// TIA Portal V17 export
// export: Created 2023-12-22T15:05:32.0644893Z, ExportSetting WithDefaults, DisplayName Totally Integrated Automation Portal, DisplayVersion V17, DisplayName TIA Portal Openness, DisplayVersion V17, DisplayName TIA Portal Version Control Interface, DisplayVersion V17, DisplayName STEP 7 Professional, DisplayVersion V17, DisplayName STEP 7 Safety, DisplayVersion V17, DisplayName WinCC Advanced, DisplayVersion V17
FUNCTION "ASCII_WCHAR_FC" : Void   // FC201, LAD
{ S7_Optimized_Access := 'TRUE' }
VERSION : 0.1
// stored: AutoNumber false, IsIECCheckEnabled false, SetENOAutomatically false, UDAEnableTagReadback false
   VAR_INPUT
      UNICODE : WChar;
   END_VAR
   VAR_OUTPUT
      ASCII_HEX : Byte;
   END_VAR
   VAR_IN_OUT
      DONE : Bool;
   END_VAR
BEGIN

REGION Network 1
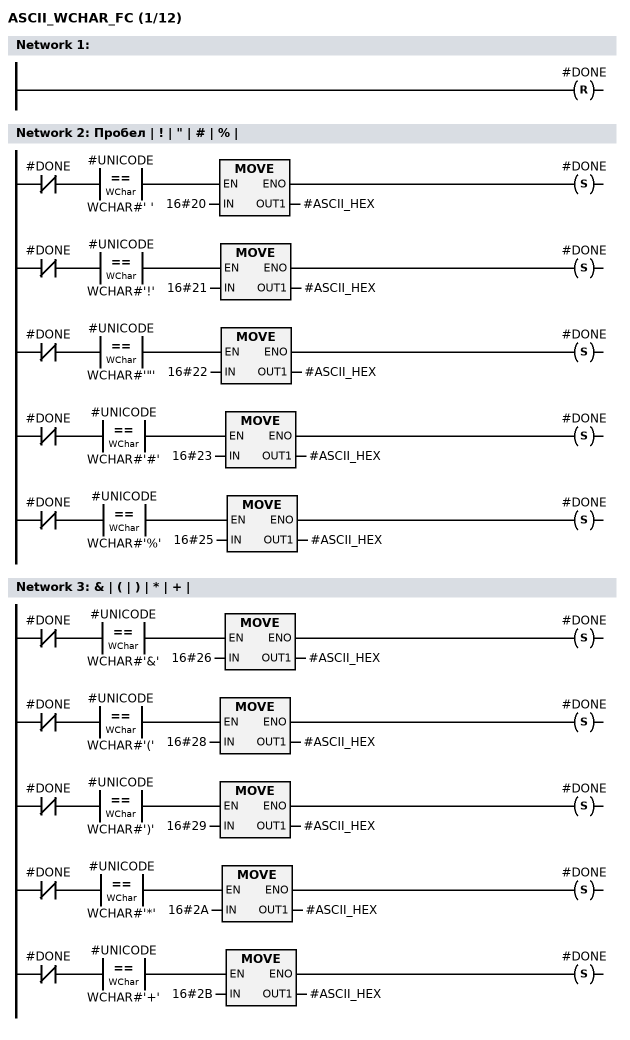
   RUNG wire#powerrail
      R_Coil( #DONE )
   END_RUNG
   // the same network as SCL:
   #DONE := FALSE;
END_REGION

REGION Network 2: Пробел | ! | " | # | % |
   RUNG wire#powerrail
      I_Contact( #DONE )
      { S7_Templates := "SrcType := WChar" } EQ_Contact(in1 := #UNICODE, in2 := WCHAR#' ')
      Move(in := 16#20, out1 => #ASCII_HEX)
      S_Coil( #DONE )
   END_RUNG
   RUNG wire#powerrail
      I_Contact( #DONE )
      { S7_Templates := "SrcType := WChar" } EQ_Contact(in1 := #UNICODE, in2 := WCHAR#'!')
      Move(in := 16#21, out1 => #ASCII_HEX)
      S_Coil( #DONE )
   END_RUNG
   RUNG wire#powerrail
      I_Contact( #DONE )
      { S7_Templates := "SrcType := WChar" } EQ_Contact(in1 := #UNICODE, in2 := WCHAR#'"')
      Move(in := 16#22, out1 => #ASCII_HEX)
      S_Coil( #DONE )
   END_RUNG
   RUNG wire#powerrail
      I_Contact( #DONE )
      { S7_Templates := "SrcType := WChar" } EQ_Contact(in1 := #UNICODE, in2 := WCHAR#'#')
      Move(in := 16#23, out1 => #ASCII_HEX)
      S_Coil( #DONE )
   END_RUNG
   RUNG wire#powerrail
      I_Contact( #DONE )
      { S7_Templates := "SrcType := WChar" } EQ_Contact(in1 := #UNICODE, in2 := WCHAR#'%')
      Move(in := 16#25, out1 => #ASCII_HEX)
      S_Coil( #DONE )
   END_RUNG
   // the same network as SCL:
   IF NOT #DONE AND (#UNICODE = WCHAR#' ') THEN
       #ASCII_HEX := 16#20;
       #DONE := TRUE;
   END_IF;
   IF NOT #DONE AND (#UNICODE = WCHAR#'!') THEN
       #ASCII_HEX := 16#21;
       #DONE := TRUE;
   END_IF;
   IF NOT #DONE AND (#UNICODE = WCHAR#'"') THEN
       #ASCII_HEX := 16#22;
       #DONE := TRUE;
   END_IF;
   IF NOT #DONE AND (#UNICODE = WCHAR#'#') THEN
       #ASCII_HEX := 16#23;
       #DONE := TRUE;
   END_IF;
   IF NOT #DONE AND (#UNICODE = WCHAR#'%') THEN
       #ASCII_HEX := 16#25;
       #DONE := TRUE;
   END_IF;
END_REGION

REGION Network 3: & | ( | ) | * | + |
   RUNG wire#powerrail
      I_Contact( #DONE )
      { S7_Templates := "SrcType := WChar" } EQ_Contact(in1 := #UNICODE, in2 := WCHAR#'&')
      Move(in := 16#26, out1 => #ASCII_HEX)
      S_Coil( #DONE )
   END_RUNG
   RUNG wire#powerrail
      I_Contact( #DONE )
      { S7_Templates := "SrcType := WChar" } EQ_Contact(in1 := #UNICODE, in2 := WCHAR#'(')
      Move(in := 16#28, out1 => #ASCII_HEX)
      S_Coil( #DONE )
   END_RUNG
   RUNG wire#powerrail
      I_Contact( #DONE )
      { S7_Templates := "SrcType := WChar" } EQ_Contact(in1 := #UNICODE, in2 := WCHAR#')')
      Move(in := 16#29, out1 => #ASCII_HEX)
      S_Coil( #DONE )
   END_RUNG
   RUNG wire#powerrail
      I_Contact( #DONE )
      { S7_Templates := "SrcType := WChar" } EQ_Contact(in1 := #UNICODE, in2 := WCHAR#'*')
      Move(in := 16#2A, out1 => #ASCII_HEX)
      S_Coil( #DONE )
   END_RUNG
   RUNG wire#powerrail
      I_Contact( #DONE )
      { S7_Templates := "SrcType := WChar" } EQ_Contact(in1 := #UNICODE, in2 := WCHAR#'+')
      Move(in := 16#2B, out1 => #ASCII_HEX)
      S_Coil( #DONE )
   END_RUNG
   // the same network as SCL:
   IF NOT #DONE AND (#UNICODE = WCHAR#'&') THEN
       #ASCII_HEX := 16#26;
       #DONE := TRUE;
   END_IF;
   IF NOT #DONE AND (#UNICODE = WCHAR#'(') THEN
       #ASCII_HEX := 16#28;
       #DONE := TRUE;
   END_IF;
   IF NOT #DONE AND (#UNICODE = WCHAR#')') THEN
       #ASCII_HEX := 16#29;
       #DONE := TRUE;
   END_IF;
   IF NOT #DONE AND (#UNICODE = WCHAR#'*') THEN
       #ASCII_HEX := 16#2A;
       #DONE := TRUE;
   END_IF;
   IF NOT #DONE AND (#UNICODE = WCHAR#'+') THEN
       #ASCII_HEX := 16#2B;
       #DONE := TRUE;
   END_IF;
END_REGION

REGION Network 4: , | - | . | / | : |
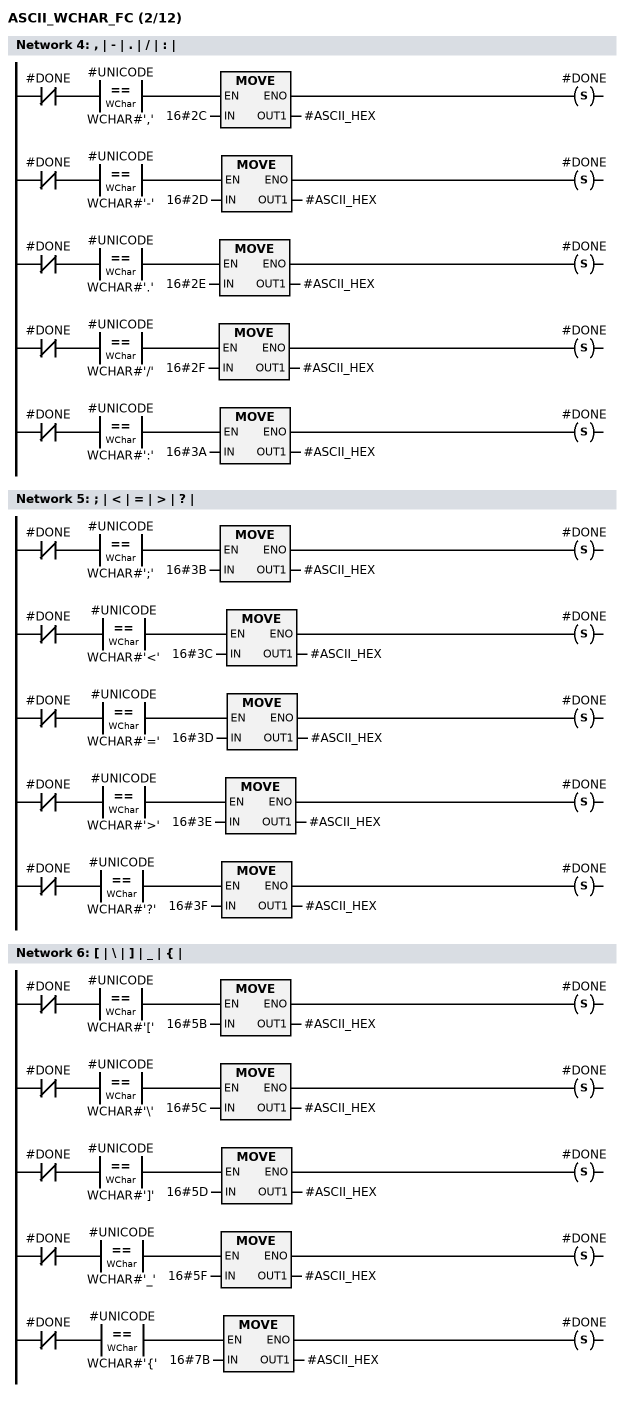
   RUNG wire#powerrail
      I_Contact( #DONE )
      { S7_Templates := "SrcType := WChar" } EQ_Contact(in1 := #UNICODE, in2 := WCHAR#',')
      Move(in := 16#2C, out1 => #ASCII_HEX)
      S_Coil( #DONE )
   END_RUNG
   RUNG wire#powerrail
      I_Contact( #DONE )
      { S7_Templates := "SrcType := WChar" } EQ_Contact(in1 := #UNICODE, in2 := WCHAR#'-')
      Move(in := 16#2D, out1 => #ASCII_HEX)
      S_Coil( #DONE )
   END_RUNG
   RUNG wire#powerrail
      I_Contact( #DONE )
      { S7_Templates := "SrcType := WChar" } EQ_Contact(in1 := #UNICODE, in2 := WCHAR#'.')
      Move(in := 16#2E, out1 => #ASCII_HEX)
      S_Coil( #DONE )
   END_RUNG
   RUNG wire#powerrail
      I_Contact( #DONE )
      { S7_Templates := "SrcType := WChar" } EQ_Contact(in1 := #UNICODE, in2 := WCHAR#'/')
      Move(in := 16#2F, out1 => #ASCII_HEX)
      S_Coil( #DONE )
   END_RUNG
   RUNG wire#powerrail
      I_Contact( #DONE )
      { S7_Templates := "SrcType := WChar" } EQ_Contact(in1 := #UNICODE, in2 := WCHAR#':')
      Move(in := 16#3A, out1 => #ASCII_HEX)
      S_Coil( #DONE )
   END_RUNG
   // the same network as SCL:
   IF NOT #DONE AND (#UNICODE = WCHAR#',') THEN
       #ASCII_HEX := 16#2C;
       #DONE := TRUE;
   END_IF;
   IF NOT #DONE AND (#UNICODE = WCHAR#'-') THEN
       #ASCII_HEX := 16#2D;
       #DONE := TRUE;
   END_IF;
   IF NOT #DONE AND (#UNICODE = WCHAR#'.') THEN
       #ASCII_HEX := 16#2E;
       #DONE := TRUE;
   END_IF;
   IF NOT #DONE AND (#UNICODE = WCHAR#'/') THEN
       #ASCII_HEX := 16#2F;
       #DONE := TRUE;
   END_IF;
   IF NOT #DONE AND (#UNICODE = WCHAR#':') THEN
       #ASCII_HEX := 16#3A;
       #DONE := TRUE;
   END_IF;
END_REGION

REGION Network 5: ; | < | = | > | ? |
   RUNG wire#powerrail
      I_Contact( #DONE )
      { S7_Templates := "SrcType := WChar" } EQ_Contact(in1 := #UNICODE, in2 := WCHAR#';')
      Move(in := 16#3B, out1 => #ASCII_HEX)
      S_Coil( #DONE )
   END_RUNG
   RUNG wire#powerrail
      I_Contact( #DONE )
      { S7_Templates := "SrcType := WChar" } EQ_Contact(in1 := #UNICODE, in2 := WCHAR#'<')
      Move(in := 16#3C, out1 => #ASCII_HEX)
      S_Coil( #DONE )
   END_RUNG
   RUNG wire#powerrail
      I_Contact( #DONE )
      { S7_Templates := "SrcType := WChar" } EQ_Contact(in1 := #UNICODE, in2 := WCHAR#'=')
      Move(in := 16#3D, out1 => #ASCII_HEX)
      S_Coil( #DONE )
   END_RUNG
   RUNG wire#powerrail
      I_Contact( #DONE )
      { S7_Templates := "SrcType := WChar" } EQ_Contact(in1 := #UNICODE, in2 := WCHAR#'>')
      Move(in := 16#3E, out1 => #ASCII_HEX)
      S_Coil( #DONE )
   END_RUNG
   RUNG wire#powerrail
      I_Contact( #DONE )
      { S7_Templates := "SrcType := WChar" } EQ_Contact(in1 := #UNICODE, in2 := WCHAR#'?')
      Move(in := 16#3F, out1 => #ASCII_HEX)
      S_Coil( #DONE )
   END_RUNG
   // the same network as SCL:
   IF NOT #DONE AND (#UNICODE = WCHAR#';') THEN
       #ASCII_HEX := 16#3B;
       #DONE := TRUE;
   END_IF;
   IF NOT #DONE AND (#UNICODE = WCHAR#'<') THEN
       #ASCII_HEX := 16#3C;
       #DONE := TRUE;
   END_IF;
   IF NOT #DONE AND (#UNICODE = WCHAR#'=') THEN
       #ASCII_HEX := 16#3D;
       #DONE := TRUE;
   END_IF;
   IF NOT #DONE AND (#UNICODE = WCHAR#'>') THEN
       #ASCII_HEX := 16#3E;
       #DONE := TRUE;
   END_IF;
   IF NOT #DONE AND (#UNICODE = WCHAR#'?') THEN
       #ASCII_HEX := 16#3F;
       #DONE := TRUE;
   END_IF;
END_REGION

REGION Network 6: [ | \ | ] | _ | { |
   RUNG wire#powerrail
      I_Contact( #DONE )
      { S7_Templates := "SrcType := WChar" } EQ_Contact(in1 := #UNICODE, in2 := WCHAR#'[')
      Move(in := 16#5B, out1 => #ASCII_HEX)
      S_Coil( #DONE )
   END_RUNG
   RUNG wire#powerrail
      I_Contact( #DONE )
      { S7_Templates := "SrcType := WChar" } EQ_Contact(in1 := #UNICODE, in2 := WCHAR#'\')
      Move(in := 16#5C, out1 => #ASCII_HEX)
      S_Coil( #DONE )
   END_RUNG
   RUNG wire#powerrail
      I_Contact( #DONE )
      { S7_Templates := "SrcType := WChar" } EQ_Contact(in1 := #UNICODE, in2 := WCHAR#']')
      Move(in := 16#5D, out1 => #ASCII_HEX)
      S_Coil( #DONE )
   END_RUNG
   RUNG wire#powerrail
      I_Contact( #DONE )
      { S7_Templates := "SrcType := WChar" } EQ_Contact(in1 := #UNICODE, in2 := WCHAR#'_')
      Move(in := 16#5F, out1 => #ASCII_HEX)
      S_Coil( #DONE )
   END_RUNG
   RUNG wire#powerrail
      I_Contact( #DONE )
      { S7_Templates := "SrcType := WChar" } EQ_Contact(in1 := #UNICODE, in2 := WCHAR#'{')
      Move(in := 16#7B, out1 => #ASCII_HEX)
      S_Coil( #DONE )
   END_RUNG
   // the same network as SCL:
   IF NOT #DONE AND (#UNICODE = WCHAR#'[') THEN
       #ASCII_HEX := 16#5B;
       #DONE := TRUE;
   END_IF;
   IF NOT #DONE AND (#UNICODE = WCHAR#'\') THEN
       #ASCII_HEX := 16#5C;
       #DONE := TRUE;
   END_IF;
   IF NOT #DONE AND (#UNICODE = WCHAR#']') THEN
       #ASCII_HEX := 16#5D;
       #DONE := TRUE;
   END_IF;
   IF NOT #DONE AND (#UNICODE = WCHAR#'_') THEN
       #ASCII_HEX := 16#5F;
       #DONE := TRUE;
   END_IF;
   IF NOT #DONE AND (#UNICODE = WCHAR#'{') THEN
       #ASCII_HEX := 16#7B;
       #DONE := TRUE;
   END_IF;
END_REGION

REGION Network 7: } | | |
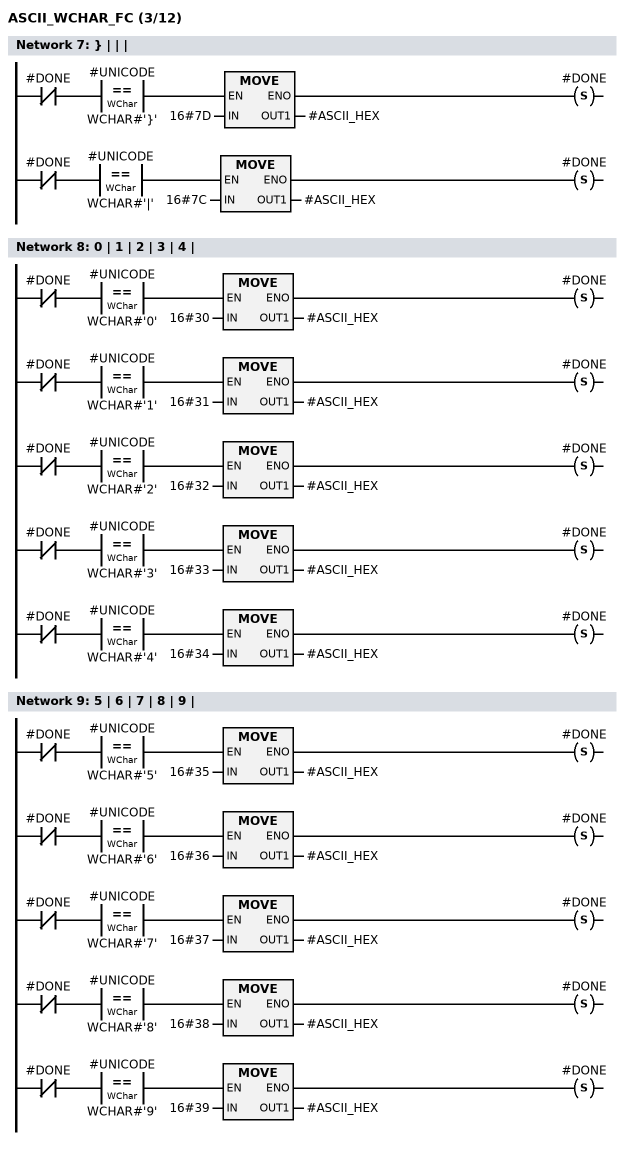
   RUNG wire#powerrail
      I_Contact( #DONE )
      { S7_Templates := "SrcType := WChar" } EQ_Contact(in1 := #UNICODE, in2 := WCHAR#'}')
      Move(in := 16#7D, out1 => #ASCII_HEX)
      S_Coil( #DONE )
   END_RUNG
   RUNG wire#powerrail
      I_Contact( #DONE )
      { S7_Templates := "SrcType := WChar" } EQ_Contact(in1 := #UNICODE, in2 := WCHAR#'|')
      Move(in := 16#7C, out1 => #ASCII_HEX)
      S_Coil( #DONE )
   END_RUNG
   // the same network as SCL:
   IF NOT #DONE AND (#UNICODE = WCHAR#'}') THEN
       #ASCII_HEX := 16#7D;
       #DONE := TRUE;
   END_IF;
   IF NOT #DONE AND (#UNICODE = WCHAR#'|') THEN
       #ASCII_HEX := 16#7C;
       #DONE := TRUE;
   END_IF;
END_REGION

REGION Network 8: 0 | 1 | 2 | 3 | 4 |
   RUNG wire#powerrail
      I_Contact( #DONE )
      { S7_Templates := "SrcType := WChar" } EQ_Contact(in1 := #UNICODE, in2 := WCHAR#'0')
      Move(in := 16#30, out1 => #ASCII_HEX)
      S_Coil( #DONE )
   END_RUNG
   RUNG wire#powerrail
      I_Contact( #DONE )
      { S7_Templates := "SrcType := WChar" } EQ_Contact(in1 := #UNICODE, in2 := WCHAR#'1')
      Move(in := 16#31, out1 => #ASCII_HEX)
      S_Coil( #DONE )
   END_RUNG
   RUNG wire#powerrail
      I_Contact( #DONE )
      { S7_Templates := "SrcType := WChar" } EQ_Contact(in1 := #UNICODE, in2 := WCHAR#'2')
      Move(in := 16#32, out1 => #ASCII_HEX)
      S_Coil( #DONE )
   END_RUNG
   RUNG wire#powerrail
      I_Contact( #DONE )
      { S7_Templates := "SrcType := WChar" } EQ_Contact(in1 := #UNICODE, in2 := WCHAR#'3')
      Move(in := 16#33, out1 => #ASCII_HEX)
      S_Coil( #DONE )
   END_RUNG
   RUNG wire#powerrail
      I_Contact( #DONE )
      { S7_Templates := "SrcType := WChar" } EQ_Contact(in1 := #UNICODE, in2 := WCHAR#'4')
      Move(in := 16#34, out1 => #ASCII_HEX)
      S_Coil( #DONE )
   END_RUNG
   // the same network as SCL:
   IF NOT #DONE AND (#UNICODE = WCHAR#'0') THEN
       #ASCII_HEX := 16#30;
       #DONE := TRUE;
   END_IF;
   IF NOT #DONE AND (#UNICODE = WCHAR#'1') THEN
       #ASCII_HEX := 16#31;
       #DONE := TRUE;
   END_IF;
   IF NOT #DONE AND (#UNICODE = WCHAR#'2') THEN
       #ASCII_HEX := 16#32;
       #DONE := TRUE;
   END_IF;
   IF NOT #DONE AND (#UNICODE = WCHAR#'3') THEN
       #ASCII_HEX := 16#33;
       #DONE := TRUE;
   END_IF;
   IF NOT #DONE AND (#UNICODE = WCHAR#'4') THEN
       #ASCII_HEX := 16#34;
       #DONE := TRUE;
   END_IF;
END_REGION

REGION Network 9: 5 | 6 | 7 | 8 | 9 |
   RUNG wire#powerrail
      I_Contact( #DONE )
      { S7_Templates := "SrcType := WChar" } EQ_Contact(in1 := #UNICODE, in2 := WCHAR#'5')
      Move(in := 16#35, out1 => #ASCII_HEX)
      S_Coil( #DONE )
   END_RUNG
   RUNG wire#powerrail
      I_Contact( #DONE )
      { S7_Templates := "SrcType := WChar" } EQ_Contact(in1 := #UNICODE, in2 := WCHAR#'6')
      Move(in := 16#36, out1 => #ASCII_HEX)
      S_Coil( #DONE )
   END_RUNG
   RUNG wire#powerrail
      I_Contact( #DONE )
      { S7_Templates := "SrcType := WChar" } EQ_Contact(in1 := #UNICODE, in2 := WCHAR#'7')
      Move(in := 16#37, out1 => #ASCII_HEX)
      S_Coil( #DONE )
   END_RUNG
   RUNG wire#powerrail
      I_Contact( #DONE )
      { S7_Templates := "SrcType := WChar" } EQ_Contact(in1 := #UNICODE, in2 := WCHAR#'8')
      Move(in := 16#38, out1 => #ASCII_HEX)
      S_Coil( #DONE )
   END_RUNG
   RUNG wire#powerrail
      I_Contact( #DONE )
      { S7_Templates := "SrcType := WChar" } EQ_Contact(in1 := #UNICODE, in2 := WCHAR#'9')
      Move(in := 16#39, out1 => #ASCII_HEX)
      S_Coil( #DONE )
   END_RUNG
   // the same network as SCL:
   IF NOT #DONE AND (#UNICODE = WCHAR#'5') THEN
       #ASCII_HEX := 16#35;
       #DONE := TRUE;
   END_IF;
   IF NOT #DONE AND (#UNICODE = WCHAR#'6') THEN
       #ASCII_HEX := 16#36;
       #DONE := TRUE;
   END_IF;
   IF NOT #DONE AND (#UNICODE = WCHAR#'7') THEN
       #ASCII_HEX := 16#37;
       #DONE := TRUE;
   END_IF;
   IF NOT #DONE AND (#UNICODE = WCHAR#'8') THEN
       #ASCII_HEX := 16#38;
       #DONE := TRUE;
   END_IF;
   IF NOT #DONE AND (#UNICODE = WCHAR#'9') THEN
       #ASCII_HEX := 16#39;
       #DONE := TRUE;
   END_IF;
END_REGION

REGION Network 10: А | Б | В | Г | Д |
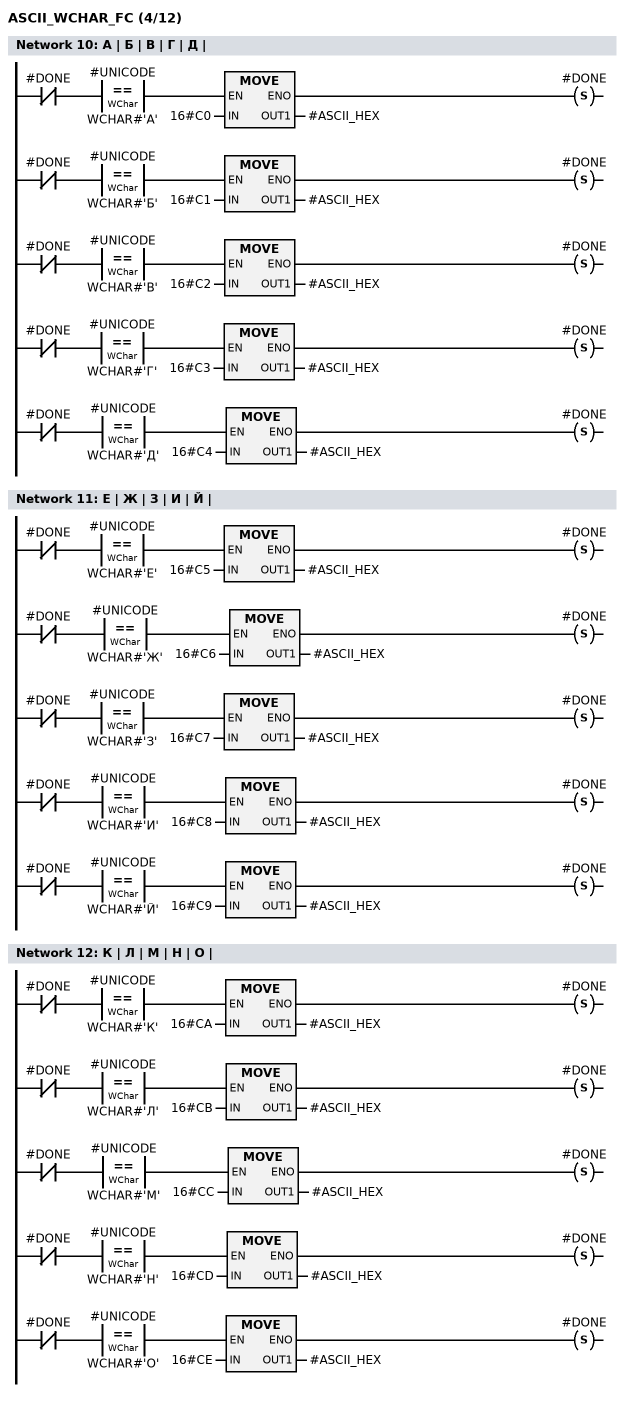
   RUNG wire#powerrail
      I_Contact( #DONE )
      { S7_Templates := "SrcType := WChar" } EQ_Contact(in1 := #UNICODE, in2 := WCHAR#'А')
      Move(in := 16#C0, out1 => #ASCII_HEX)
      S_Coil( #DONE )
   END_RUNG
   RUNG wire#powerrail
      I_Contact( #DONE )
      { S7_Templates := "SrcType := WChar" } EQ_Contact(in1 := #UNICODE, in2 := WCHAR#'Б')
      Move(in := 16#C1, out1 => #ASCII_HEX)
      S_Coil( #DONE )
   END_RUNG
   RUNG wire#powerrail
      I_Contact( #DONE )
      { S7_Templates := "SrcType := WChar" } EQ_Contact(in1 := #UNICODE, in2 := WCHAR#'В')
      Move(in := 16#C2, out1 => #ASCII_HEX)
      S_Coil( #DONE )
   END_RUNG
   RUNG wire#powerrail
      I_Contact( #DONE )
      { S7_Templates := "SrcType := WChar" } EQ_Contact(in1 := #UNICODE, in2 := WCHAR#'Г')
      Move(in := 16#C3, out1 => #ASCII_HEX)
      S_Coil( #DONE )
   END_RUNG
   RUNG wire#powerrail
      I_Contact( #DONE )
      { S7_Templates := "SrcType := WChar" } EQ_Contact(in1 := #UNICODE, in2 := WCHAR#'Д')
      Move(in := 16#C4, out1 => #ASCII_HEX)
      S_Coil( #DONE )
   END_RUNG
   // the same network as SCL:
   IF NOT #DONE AND (#UNICODE = WCHAR#'А') THEN
       #ASCII_HEX := 16#C0;
       #DONE := TRUE;
   END_IF;
   IF NOT #DONE AND (#UNICODE = WCHAR#'Б') THEN
       #ASCII_HEX := 16#C1;
       #DONE := TRUE;
   END_IF;
   IF NOT #DONE AND (#UNICODE = WCHAR#'В') THEN
       #ASCII_HEX := 16#C2;
       #DONE := TRUE;
   END_IF;
   IF NOT #DONE AND (#UNICODE = WCHAR#'Г') THEN
       #ASCII_HEX := 16#C3;
       #DONE := TRUE;
   END_IF;
   IF NOT #DONE AND (#UNICODE = WCHAR#'Д') THEN
       #ASCII_HEX := 16#C4;
       #DONE := TRUE;
   END_IF;
END_REGION

REGION Network 11: Е | Ж | З | И | Й |
   RUNG wire#powerrail
      I_Contact( #DONE )
      { S7_Templates := "SrcType := WChar" } EQ_Contact(in1 := #UNICODE, in2 := WCHAR#'Е')
      Move(in := 16#C5, out1 => #ASCII_HEX)
      S_Coil( #DONE )
   END_RUNG
   RUNG wire#powerrail
      I_Contact( #DONE )
      { S7_Templates := "SrcType := WChar" } EQ_Contact(in1 := #UNICODE, in2 := WCHAR#'Ж')
      Move(in := 16#C6, out1 => #ASCII_HEX)
      S_Coil( #DONE )
   END_RUNG
   RUNG wire#powerrail
      I_Contact( #DONE )
      { S7_Templates := "SrcType := WChar" } EQ_Contact(in1 := #UNICODE, in2 := WCHAR#'З')
      Move(in := 16#C7, out1 => #ASCII_HEX)
      S_Coil( #DONE )
   END_RUNG
   RUNG wire#powerrail
      I_Contact( #DONE )
      { S7_Templates := "SrcType := WChar" } EQ_Contact(in1 := #UNICODE, in2 := WCHAR#'И')
      Move(in := 16#C8, out1 => #ASCII_HEX)
      S_Coil( #DONE )
   END_RUNG
   RUNG wire#powerrail
      I_Contact( #DONE )
      { S7_Templates := "SrcType := WChar" } EQ_Contact(in1 := #UNICODE, in2 := WCHAR#'Й')
      Move(in := 16#C9, out1 => #ASCII_HEX)
      S_Coil( #DONE )
   END_RUNG
   // the same network as SCL:
   IF NOT #DONE AND (#UNICODE = WCHAR#'Е') THEN
       #ASCII_HEX := 16#C5;
       #DONE := TRUE;
   END_IF;
   IF NOT #DONE AND (#UNICODE = WCHAR#'Ж') THEN
       #ASCII_HEX := 16#C6;
       #DONE := TRUE;
   END_IF;
   IF NOT #DONE AND (#UNICODE = WCHAR#'З') THEN
       #ASCII_HEX := 16#C7;
       #DONE := TRUE;
   END_IF;
   IF NOT #DONE AND (#UNICODE = WCHAR#'И') THEN
       #ASCII_HEX := 16#C8;
       #DONE := TRUE;
   END_IF;
   IF NOT #DONE AND (#UNICODE = WCHAR#'Й') THEN
       #ASCII_HEX := 16#C9;
       #DONE := TRUE;
   END_IF;
END_REGION

REGION Network 12: К | Л | М | Н | О |
   RUNG wire#powerrail
      I_Contact( #DONE )
      { S7_Templates := "SrcType := WChar" } EQ_Contact(in1 := #UNICODE, in2 := WCHAR#'К')
      Move(in := 16#CA, out1 => #ASCII_HEX)
      S_Coil( #DONE )
   END_RUNG
   RUNG wire#powerrail
      I_Contact( #DONE )
      { S7_Templates := "SrcType := WChar" } EQ_Contact(in1 := #UNICODE, in2 := WCHAR#'Л')
      Move(in := 16#CB, out1 => #ASCII_HEX)
      S_Coil( #DONE )
   END_RUNG
   RUNG wire#powerrail
      I_Contact( #DONE )
      { S7_Templates := "SrcType := WChar" } EQ_Contact(in1 := #UNICODE, in2 := WCHAR#'М')
      Move(in := 16#CC, out1 => #ASCII_HEX)
      S_Coil( #DONE )
   END_RUNG
   RUNG wire#powerrail
      I_Contact( #DONE )
      { S7_Templates := "SrcType := WChar" } EQ_Contact(in1 := #UNICODE, in2 := WCHAR#'Н')
      Move(in := 16#CD, out1 => #ASCII_HEX)
      S_Coil( #DONE )
   END_RUNG
   RUNG wire#powerrail
      I_Contact( #DONE )
      { S7_Templates := "SrcType := WChar" } EQ_Contact(in1 := #UNICODE, in2 := WCHAR#'О')
      Move(in := 16#CE, out1 => #ASCII_HEX)
      S_Coil( #DONE )
   END_RUNG
   // the same network as SCL:
   IF NOT #DONE AND (#UNICODE = WCHAR#'К') THEN
       #ASCII_HEX := 16#CA;
       #DONE := TRUE;
   END_IF;
   IF NOT #DONE AND (#UNICODE = WCHAR#'Л') THEN
       #ASCII_HEX := 16#CB;
       #DONE := TRUE;
   END_IF;
   IF NOT #DONE AND (#UNICODE = WCHAR#'М') THEN
       #ASCII_HEX := 16#CC;
       #DONE := TRUE;
   END_IF;
   IF NOT #DONE AND (#UNICODE = WCHAR#'Н') THEN
       #ASCII_HEX := 16#CD;
       #DONE := TRUE;
   END_IF;
   IF NOT #DONE AND (#UNICODE = WCHAR#'О') THEN
       #ASCII_HEX := 16#CE;
       #DONE := TRUE;
   END_IF;
END_REGION

REGION Network 13: П | Р | С | Т | У |
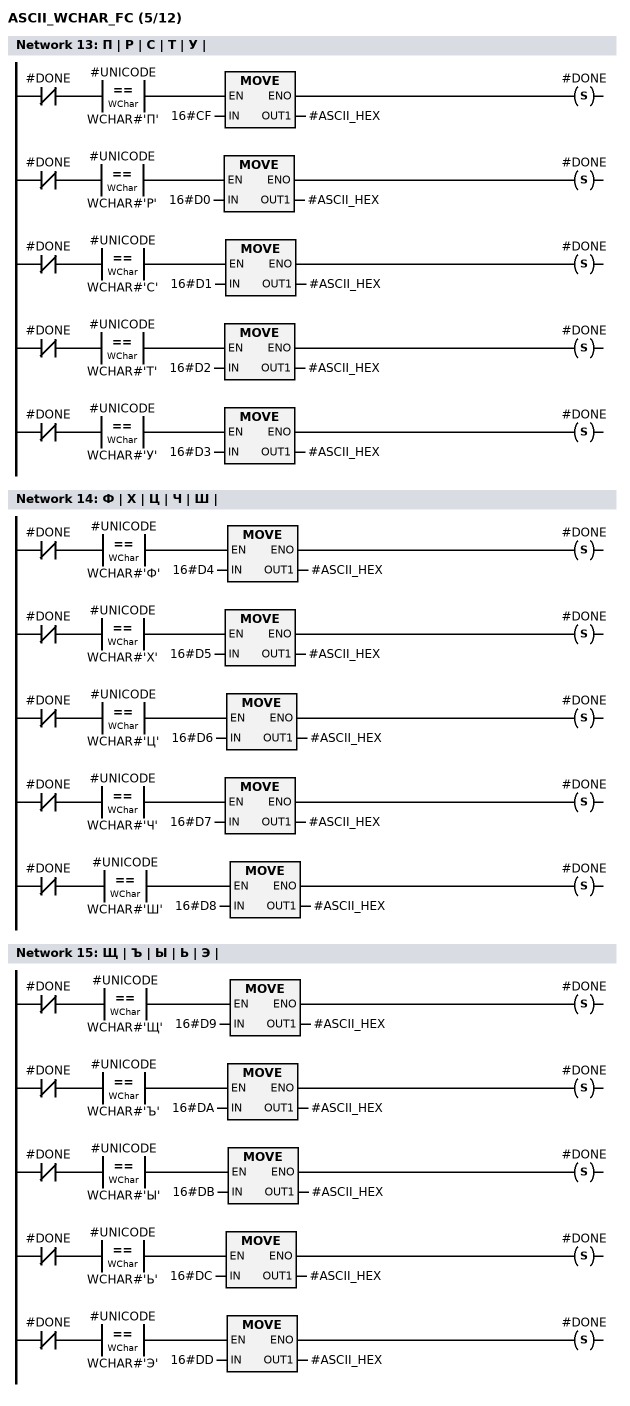
   RUNG wire#powerrail
      I_Contact( #DONE )
      { S7_Templates := "SrcType := WChar" } EQ_Contact(in1 := #UNICODE, in2 := WCHAR#'П')
      Move(in := 16#CF, out1 => #ASCII_HEX)
      S_Coil( #DONE )
   END_RUNG
   RUNG wire#powerrail
      I_Contact( #DONE )
      { S7_Templates := "SrcType := WChar" } EQ_Contact(in1 := #UNICODE, in2 := WCHAR#'Р')
      Move(in := 16#D0, out1 => #ASCII_HEX)
      S_Coil( #DONE )
   END_RUNG
   RUNG wire#powerrail
      I_Contact( #DONE )
      { S7_Templates := "SrcType := WChar" } EQ_Contact(in1 := #UNICODE, in2 := WCHAR#'С')
      Move(in := 16#D1, out1 => #ASCII_HEX)
      S_Coil( #DONE )
   END_RUNG
   RUNG wire#powerrail
      I_Contact( #DONE )
      { S7_Templates := "SrcType := WChar" } EQ_Contact(in1 := #UNICODE, in2 := WCHAR#'Т')
      Move(in := 16#D2, out1 => #ASCII_HEX)
      S_Coil( #DONE )
   END_RUNG
   RUNG wire#powerrail
      I_Contact( #DONE )
      { S7_Templates := "SrcType := WChar" } EQ_Contact(in1 := #UNICODE, in2 := WCHAR#'У')
      Move(in := 16#D3, out1 => #ASCII_HEX)
      S_Coil( #DONE )
   END_RUNG
   // the same network as SCL:
   IF NOT #DONE AND (#UNICODE = WCHAR#'П') THEN
       #ASCII_HEX := 16#CF;
       #DONE := TRUE;
   END_IF;
   IF NOT #DONE AND (#UNICODE = WCHAR#'Р') THEN
       #ASCII_HEX := 16#D0;
       #DONE := TRUE;
   END_IF;
   IF NOT #DONE AND (#UNICODE = WCHAR#'С') THEN
       #ASCII_HEX := 16#D1;
       #DONE := TRUE;
   END_IF;
   IF NOT #DONE AND (#UNICODE = WCHAR#'Т') THEN
       #ASCII_HEX := 16#D2;
       #DONE := TRUE;
   END_IF;
   IF NOT #DONE AND (#UNICODE = WCHAR#'У') THEN
       #ASCII_HEX := 16#D3;
       #DONE := TRUE;
   END_IF;
END_REGION

REGION Network 14: Ф | Х | Ц | Ч | Ш |
   RUNG wire#powerrail
      I_Contact( #DONE )
      { S7_Templates := "SrcType := WChar" } EQ_Contact(in1 := #UNICODE, in2 := WCHAR#'Ф')
      Move(in := 16#D4, out1 => #ASCII_HEX)
      S_Coil( #DONE )
   END_RUNG
   RUNG wire#powerrail
      I_Contact( #DONE )
      { S7_Templates := "SrcType := WChar" } EQ_Contact(in1 := #UNICODE, in2 := WCHAR#'Х')
      Move(in := 16#D5, out1 => #ASCII_HEX)
      S_Coil( #DONE )
   END_RUNG
   RUNG wire#powerrail
      I_Contact( #DONE )
      { S7_Templates := "SrcType := WChar" } EQ_Contact(in1 := #UNICODE, in2 := WCHAR#'Ц')
      Move(in := 16#D6, out1 => #ASCII_HEX)
      S_Coil( #DONE )
   END_RUNG
   RUNG wire#powerrail
      I_Contact( #DONE )
      { S7_Templates := "SrcType := WChar" } EQ_Contact(in1 := #UNICODE, in2 := WCHAR#'Ч')
      Move(in := 16#D7, out1 => #ASCII_HEX)
      S_Coil( #DONE )
   END_RUNG
   RUNG wire#powerrail
      I_Contact( #DONE )
      { S7_Templates := "SrcType := WChar" } EQ_Contact(in1 := #UNICODE, in2 := WCHAR#'Ш')
      Move(in := 16#D8, out1 => #ASCII_HEX)
      S_Coil( #DONE )
   END_RUNG
   // the same network as SCL:
   IF NOT #DONE AND (#UNICODE = WCHAR#'Ф') THEN
       #ASCII_HEX := 16#D4;
       #DONE := TRUE;
   END_IF;
   IF NOT #DONE AND (#UNICODE = WCHAR#'Х') THEN
       #ASCII_HEX := 16#D5;
       #DONE := TRUE;
   END_IF;
   IF NOT #DONE AND (#UNICODE = WCHAR#'Ц') THEN
       #ASCII_HEX := 16#D6;
       #DONE := TRUE;
   END_IF;
   IF NOT #DONE AND (#UNICODE = WCHAR#'Ч') THEN
       #ASCII_HEX := 16#D7;
       #DONE := TRUE;
   END_IF;
   IF NOT #DONE AND (#UNICODE = WCHAR#'Ш') THEN
       #ASCII_HEX := 16#D8;
       #DONE := TRUE;
   END_IF;
END_REGION

REGION Network 15: Щ | Ъ | Ы | Ь | Э |
   RUNG wire#powerrail
      I_Contact( #DONE )
      { S7_Templates := "SrcType := WChar" } EQ_Contact(in1 := #UNICODE, in2 := WCHAR#'Щ')
      Move(in := 16#D9, out1 => #ASCII_HEX)
      S_Coil( #DONE )
   END_RUNG
   RUNG wire#powerrail
      I_Contact( #DONE )
      { S7_Templates := "SrcType := WChar" } EQ_Contact(in1 := #UNICODE, in2 := WCHAR#'Ъ')
      Move(in := 16#DA, out1 => #ASCII_HEX)
      S_Coil( #DONE )
   END_RUNG
   RUNG wire#powerrail
      I_Contact( #DONE )
      { S7_Templates := "SrcType := WChar" } EQ_Contact(in1 := #UNICODE, in2 := WCHAR#'Ы')
      Move(in := 16#DB, out1 => #ASCII_HEX)
      S_Coil( #DONE )
   END_RUNG
   RUNG wire#powerrail
      I_Contact( #DONE )
      { S7_Templates := "SrcType := WChar" } EQ_Contact(in1 := #UNICODE, in2 := WCHAR#'Ь')
      Move(in := 16#DC, out1 => #ASCII_HEX)
      S_Coil( #DONE )
   END_RUNG
   RUNG wire#powerrail
      I_Contact( #DONE )
      { S7_Templates := "SrcType := WChar" } EQ_Contact(in1 := #UNICODE, in2 := WCHAR#'Э')
      Move(in := 16#DD, out1 => #ASCII_HEX)
      S_Coil( #DONE )
   END_RUNG
   // the same network as SCL:
   IF NOT #DONE AND (#UNICODE = WCHAR#'Щ') THEN
       #ASCII_HEX := 16#D9;
       #DONE := TRUE;
   END_IF;
   IF NOT #DONE AND (#UNICODE = WCHAR#'Ъ') THEN
       #ASCII_HEX := 16#DA;
       #DONE := TRUE;
   END_IF;
   IF NOT #DONE AND (#UNICODE = WCHAR#'Ы') THEN
       #ASCII_HEX := 16#DB;
       #DONE := TRUE;
   END_IF;
   IF NOT #DONE AND (#UNICODE = WCHAR#'Ь') THEN
       #ASCII_HEX := 16#DC;
       #DONE := TRUE;
   END_IF;
   IF NOT #DONE AND (#UNICODE = WCHAR#'Э') THEN
       #ASCII_HEX := 16#DD;
       #DONE := TRUE;
   END_IF;
END_REGION

REGION Network 16: Ю | Я |
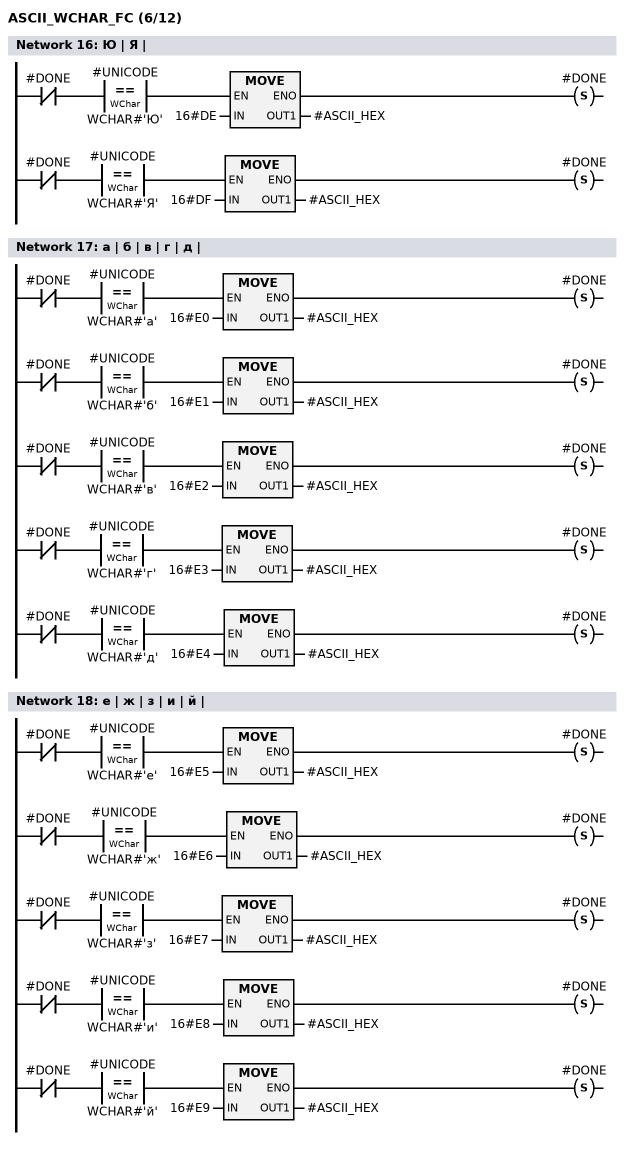
   RUNG wire#powerrail
      I_Contact( #DONE )
      { S7_Templates := "SrcType := WChar" } EQ_Contact(in1 := #UNICODE, in2 := WCHAR#'Ю')
      Move(in := 16#DE, out1 => #ASCII_HEX)
      S_Coil( #DONE )
   END_RUNG
   RUNG wire#powerrail
      I_Contact( #DONE )
      { S7_Templates := "SrcType := WChar" } EQ_Contact(in1 := #UNICODE, in2 := WCHAR#'Я')
      Move(in := 16#DF, out1 => #ASCII_HEX)
      S_Coil( #DONE )
   END_RUNG
   // the same network as SCL:
   IF NOT #DONE AND (#UNICODE = WCHAR#'Ю') THEN
       #ASCII_HEX := 16#DE;
       #DONE := TRUE;
   END_IF;
   IF NOT #DONE AND (#UNICODE = WCHAR#'Я') THEN
       #ASCII_HEX := 16#DF;
       #DONE := TRUE;
   END_IF;
END_REGION

REGION Network 17: а | б | в | г | д |
   RUNG wire#powerrail
      I_Contact( #DONE )
      { S7_Templates := "SrcType := WChar" } EQ_Contact(in1 := #UNICODE, in2 := WCHAR#'а')
      Move(in := 16#E0, out1 => #ASCII_HEX)
      S_Coil( #DONE )
   END_RUNG
   RUNG wire#powerrail
      I_Contact( #DONE )
      { S7_Templates := "SrcType := WChar" } EQ_Contact(in1 := #UNICODE, in2 := WCHAR#'б')
      Move(in := 16#E1, out1 => #ASCII_HEX)
      S_Coil( #DONE )
   END_RUNG
   RUNG wire#powerrail
      I_Contact( #DONE )
      { S7_Templates := "SrcType := WChar" } EQ_Contact(in1 := #UNICODE, in2 := WCHAR#'в')
      Move(in := 16#E2, out1 => #ASCII_HEX)
      S_Coil( #DONE )
   END_RUNG
   RUNG wire#powerrail
      I_Contact( #DONE )
      { S7_Templates := "SrcType := WChar" } EQ_Contact(in1 := #UNICODE, in2 := WCHAR#'г')
      Move(in := 16#E3, out1 => #ASCII_HEX)
      S_Coil( #DONE )
   END_RUNG
   RUNG wire#powerrail
      I_Contact( #DONE )
      { S7_Templates := "SrcType := WChar" } EQ_Contact(in1 := #UNICODE, in2 := WCHAR#'д')
      Move(in := 16#E4, out1 => #ASCII_HEX)
      S_Coil( #DONE )
   END_RUNG
   // the same network as SCL:
   IF NOT #DONE AND (#UNICODE = WCHAR#'а') THEN
       #ASCII_HEX := 16#E0;
       #DONE := TRUE;
   END_IF;
   IF NOT #DONE AND (#UNICODE = WCHAR#'б') THEN
       #ASCII_HEX := 16#E1;
       #DONE := TRUE;
   END_IF;
   IF NOT #DONE AND (#UNICODE = WCHAR#'в') THEN
       #ASCII_HEX := 16#E2;
       #DONE := TRUE;
   END_IF;
   IF NOT #DONE AND (#UNICODE = WCHAR#'г') THEN
       #ASCII_HEX := 16#E3;
       #DONE := TRUE;
   END_IF;
   IF NOT #DONE AND (#UNICODE = WCHAR#'д') THEN
       #ASCII_HEX := 16#E4;
       #DONE := TRUE;
   END_IF;
END_REGION

REGION Network 18: е | ж | з | и | й |
   RUNG wire#powerrail
      I_Contact( #DONE )
      { S7_Templates := "SrcType := WChar" } EQ_Contact(in1 := #UNICODE, in2 := WCHAR#'е')
      Move(in := 16#E5, out1 => #ASCII_HEX)
      S_Coil( #DONE )
   END_RUNG
   RUNG wire#powerrail
      I_Contact( #DONE )
      { S7_Templates := "SrcType := WChar" } EQ_Contact(in1 := #UNICODE, in2 := WCHAR#'ж')
      Move(in := 16#E6, out1 => #ASCII_HEX)
      S_Coil( #DONE )
   END_RUNG
   RUNG wire#powerrail
      I_Contact( #DONE )
      { S7_Templates := "SrcType := WChar" } EQ_Contact(in1 := #UNICODE, in2 := WCHAR#'з')
      Move(in := 16#E7, out1 => #ASCII_HEX)
      S_Coil( #DONE )
   END_RUNG
   RUNG wire#powerrail
      I_Contact( #DONE )
      { S7_Templates := "SrcType := WChar" } EQ_Contact(in1 := #UNICODE, in2 := WCHAR#'и')
      Move(in := 16#E8, out1 => #ASCII_HEX)
      S_Coil( #DONE )
   END_RUNG
   RUNG wire#powerrail
      I_Contact( #DONE )
      { S7_Templates := "SrcType := WChar" } EQ_Contact(in1 := #UNICODE, in2 := WCHAR#'й')
      Move(in := 16#E9, out1 => #ASCII_HEX)
      S_Coil( #DONE )
   END_RUNG
   // the same network as SCL:
   IF NOT #DONE AND (#UNICODE = WCHAR#'е') THEN
       #ASCII_HEX := 16#E5;
       #DONE := TRUE;
   END_IF;
   IF NOT #DONE AND (#UNICODE = WCHAR#'ж') THEN
       #ASCII_HEX := 16#E6;
       #DONE := TRUE;
   END_IF;
   IF NOT #DONE AND (#UNICODE = WCHAR#'з') THEN
       #ASCII_HEX := 16#E7;
       #DONE := TRUE;
   END_IF;
   IF NOT #DONE AND (#UNICODE = WCHAR#'и') THEN
       #ASCII_HEX := 16#E8;
       #DONE := TRUE;
   END_IF;
   IF NOT #DONE AND (#UNICODE = WCHAR#'й') THEN
       #ASCII_HEX := 16#E9;
       #DONE := TRUE;
   END_IF;
END_REGION

REGION Network 19: к | л | м | н | о |
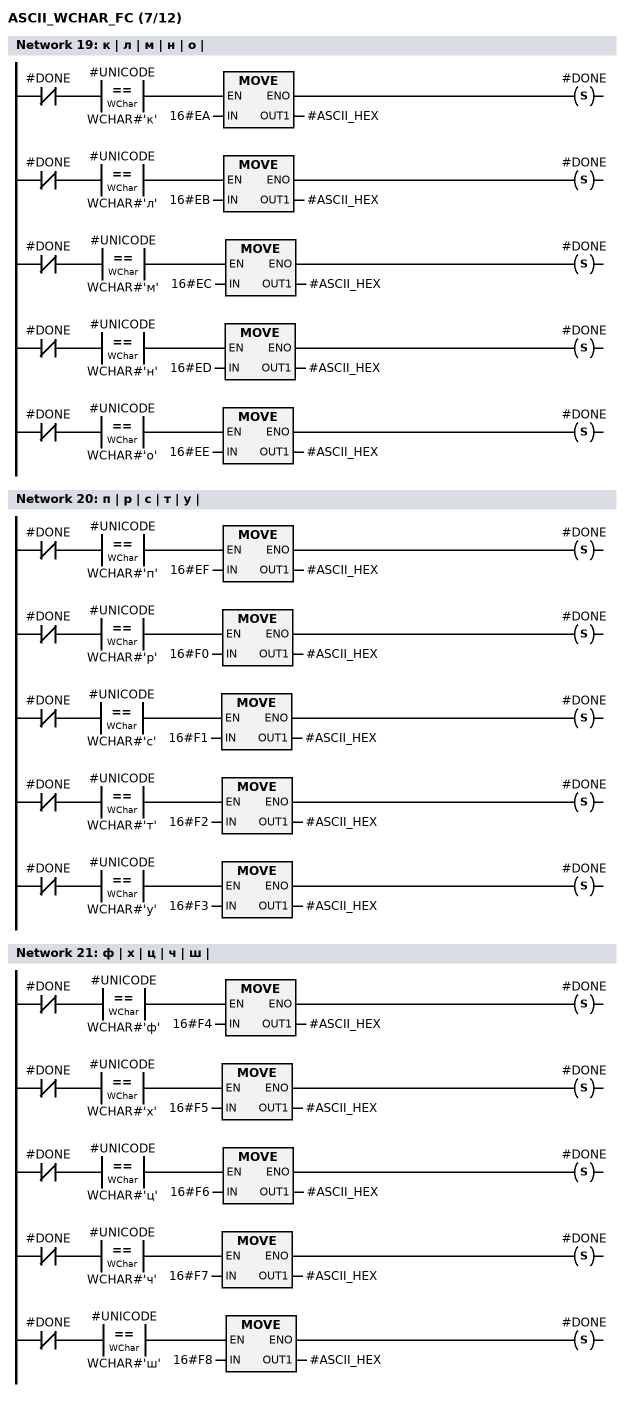
   RUNG wire#powerrail
      I_Contact( #DONE )
      { S7_Templates := "SrcType := WChar" } EQ_Contact(in1 := #UNICODE, in2 := WCHAR#'к')
      Move(in := 16#EA, out1 => #ASCII_HEX)
      S_Coil( #DONE )
   END_RUNG
   RUNG wire#powerrail
      I_Contact( #DONE )
      { S7_Templates := "SrcType := WChar" } EQ_Contact(in1 := #UNICODE, in2 := WCHAR#'л')
      Move(in := 16#EB, out1 => #ASCII_HEX)
      S_Coil( #DONE )
   END_RUNG
   RUNG wire#powerrail
      I_Contact( #DONE )
      { S7_Templates := "SrcType := WChar" } EQ_Contact(in1 := #UNICODE, in2 := WCHAR#'м')
      Move(in := 16#EC, out1 => #ASCII_HEX)
      S_Coil( #DONE )
   END_RUNG
   RUNG wire#powerrail
      I_Contact( #DONE )
      { S7_Templates := "SrcType := WChar" } EQ_Contact(in1 := #UNICODE, in2 := WCHAR#'н')
      Move(in := 16#ED, out1 => #ASCII_HEX)
      S_Coil( #DONE )
   END_RUNG
   RUNG wire#powerrail
      I_Contact( #DONE )
      { S7_Templates := "SrcType := WChar" } EQ_Contact(in1 := #UNICODE, in2 := WCHAR#'о')
      Move(in := 16#EE, out1 => #ASCII_HEX)
      S_Coil( #DONE )
   END_RUNG
   // the same network as SCL:
   IF NOT #DONE AND (#UNICODE = WCHAR#'к') THEN
       #ASCII_HEX := 16#EA;
       #DONE := TRUE;
   END_IF;
   IF NOT #DONE AND (#UNICODE = WCHAR#'л') THEN
       #ASCII_HEX := 16#EB;
       #DONE := TRUE;
   END_IF;
   IF NOT #DONE AND (#UNICODE = WCHAR#'м') THEN
       #ASCII_HEX := 16#EC;
       #DONE := TRUE;
   END_IF;
   IF NOT #DONE AND (#UNICODE = WCHAR#'н') THEN
       #ASCII_HEX := 16#ED;
       #DONE := TRUE;
   END_IF;
   IF NOT #DONE AND (#UNICODE = WCHAR#'о') THEN
       #ASCII_HEX := 16#EE;
       #DONE := TRUE;
   END_IF;
END_REGION

REGION Network 20: п | р | с | т | у |
   RUNG wire#powerrail
      I_Contact( #DONE )
      { S7_Templates := "SrcType := WChar" } EQ_Contact(in1 := #UNICODE, in2 := WCHAR#'п')
      Move(in := 16#EF, out1 => #ASCII_HEX)
      S_Coil( #DONE )
   END_RUNG
   RUNG wire#powerrail
      I_Contact( #DONE )
      { S7_Templates := "SrcType := WChar" } EQ_Contact(in1 := #UNICODE, in2 := WCHAR#'р')
      Move(in := 16#F0, out1 => #ASCII_HEX)
      S_Coil( #DONE )
   END_RUNG
   RUNG wire#powerrail
      I_Contact( #DONE )
      { S7_Templates := "SrcType := WChar" } EQ_Contact(in1 := #UNICODE, in2 := WCHAR#'с')
      Move(in := 16#F1, out1 => #ASCII_HEX)
      S_Coil( #DONE )
   END_RUNG
   RUNG wire#powerrail
      I_Contact( #DONE )
      { S7_Templates := "SrcType := WChar" } EQ_Contact(in1 := #UNICODE, in2 := WCHAR#'т')
      Move(in := 16#F2, out1 => #ASCII_HEX)
      S_Coil( #DONE )
   END_RUNG
   RUNG wire#powerrail
      I_Contact( #DONE )
      { S7_Templates := "SrcType := WChar" } EQ_Contact(in1 := #UNICODE, in2 := WCHAR#'у')
      Move(in := 16#F3, out1 => #ASCII_HEX)
      S_Coil( #DONE )
   END_RUNG
   // the same network as SCL:
   IF NOT #DONE AND (#UNICODE = WCHAR#'п') THEN
       #ASCII_HEX := 16#EF;
       #DONE := TRUE;
   END_IF;
   IF NOT #DONE AND (#UNICODE = WCHAR#'р') THEN
       #ASCII_HEX := 16#F0;
       #DONE := TRUE;
   END_IF;
   IF NOT #DONE AND (#UNICODE = WCHAR#'с') THEN
       #ASCII_HEX := 16#F1;
       #DONE := TRUE;
   END_IF;
   IF NOT #DONE AND (#UNICODE = WCHAR#'т') THEN
       #ASCII_HEX := 16#F2;
       #DONE := TRUE;
   END_IF;
   IF NOT #DONE AND (#UNICODE = WCHAR#'у') THEN
       #ASCII_HEX := 16#F3;
       #DONE := TRUE;
   END_IF;
END_REGION

REGION Network 21: ф | х | ц | ч | ш |
   RUNG wire#powerrail
      I_Contact( #DONE )
      { S7_Templates := "SrcType := WChar" } EQ_Contact(in1 := #UNICODE, in2 := WCHAR#'ф')
      Move(in := 16#F4, out1 => #ASCII_HEX)
      S_Coil( #DONE )
   END_RUNG
   RUNG wire#powerrail
      I_Contact( #DONE )
      { S7_Templates := "SrcType := WChar" } EQ_Contact(in1 := #UNICODE, in2 := WCHAR#'х')
      Move(in := 16#F5, out1 => #ASCII_HEX)
      S_Coil( #DONE )
   END_RUNG
   RUNG wire#powerrail
      I_Contact( #DONE )
      { S7_Templates := "SrcType := WChar" } EQ_Contact(in1 := #UNICODE, in2 := WCHAR#'ц')
      Move(in := 16#F6, out1 => #ASCII_HEX)
      S_Coil( #DONE )
   END_RUNG
   RUNG wire#powerrail
      I_Contact( #DONE )
      { S7_Templates := "SrcType := WChar" } EQ_Contact(in1 := #UNICODE, in2 := WCHAR#'ч')
      Move(in := 16#F7, out1 => #ASCII_HEX)
      S_Coil( #DONE )
   END_RUNG
   RUNG wire#powerrail
      I_Contact( #DONE )
      { S7_Templates := "SrcType := WChar" } EQ_Contact(in1 := #UNICODE, in2 := WCHAR#'ш')
      Move(in := 16#F8, out1 => #ASCII_HEX)
      S_Coil( #DONE )
   END_RUNG
   // the same network as SCL:
   IF NOT #DONE AND (#UNICODE = WCHAR#'ф') THEN
       #ASCII_HEX := 16#F4;
       #DONE := TRUE;
   END_IF;
   IF NOT #DONE AND (#UNICODE = WCHAR#'х') THEN
       #ASCII_HEX := 16#F5;
       #DONE := TRUE;
   END_IF;
   IF NOT #DONE AND (#UNICODE = WCHAR#'ц') THEN
       #ASCII_HEX := 16#F6;
       #DONE := TRUE;
   END_IF;
   IF NOT #DONE AND (#UNICODE = WCHAR#'ч') THEN
       #ASCII_HEX := 16#F7;
       #DONE := TRUE;
   END_IF;
   IF NOT #DONE AND (#UNICODE = WCHAR#'ш') THEN
       #ASCII_HEX := 16#F8;
       #DONE := TRUE;
   END_IF;
END_REGION

REGION Network 22: щ | ъ | ы | ь | э |
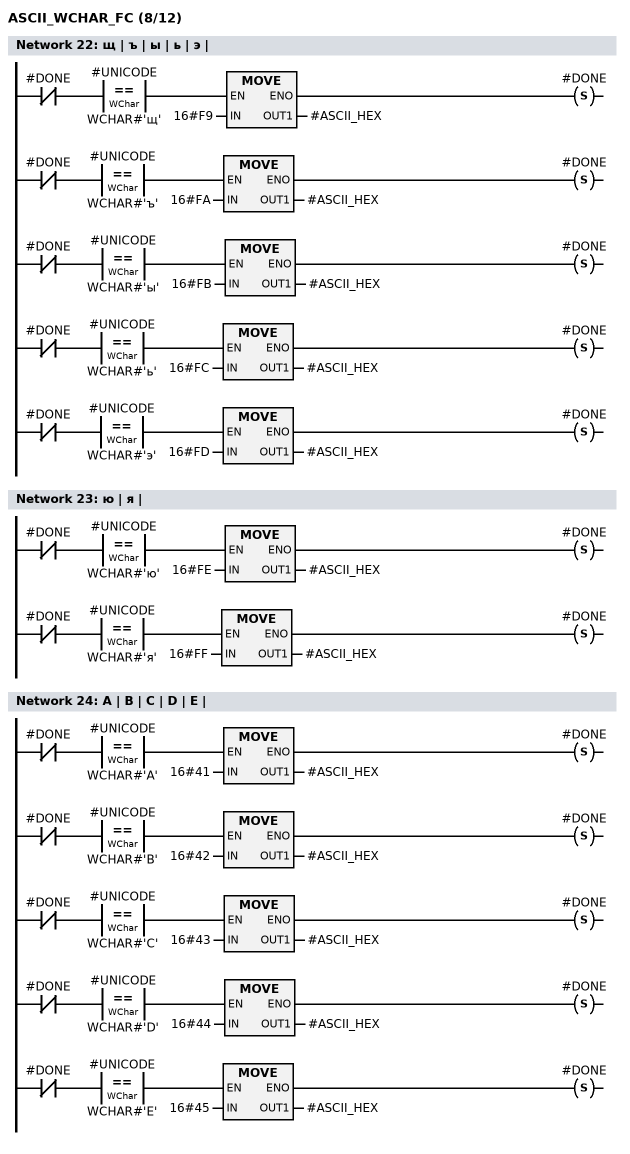
   RUNG wire#powerrail
      I_Contact( #DONE )
      { S7_Templates := "SrcType := WChar" } EQ_Contact(in1 := #UNICODE, in2 := WCHAR#'щ')
      Move(in := 16#F9, out1 => #ASCII_HEX)
      S_Coil( #DONE )
   END_RUNG
   RUNG wire#powerrail
      I_Contact( #DONE )
      { S7_Templates := "SrcType := WChar" } EQ_Contact(in1 := #UNICODE, in2 := WCHAR#'ъ')
      Move(in := 16#FA, out1 => #ASCII_HEX)
      S_Coil( #DONE )
   END_RUNG
   RUNG wire#powerrail
      I_Contact( #DONE )
      { S7_Templates := "SrcType := WChar" } EQ_Contact(in1 := #UNICODE, in2 := WCHAR#'ы')
      Move(in := 16#FB, out1 => #ASCII_HEX)
      S_Coil( #DONE )
   END_RUNG
   RUNG wire#powerrail
      I_Contact( #DONE )
      { S7_Templates := "SrcType := WChar" } EQ_Contact(in1 := #UNICODE, in2 := WCHAR#'ь')
      Move(in := 16#FC, out1 => #ASCII_HEX)
      S_Coil( #DONE )
   END_RUNG
   RUNG wire#powerrail
      I_Contact( #DONE )
      { S7_Templates := "SrcType := WChar" } EQ_Contact(in1 := #UNICODE, in2 := WCHAR#'э')
      Move(in := 16#FD, out1 => #ASCII_HEX)
      S_Coil( #DONE )
   END_RUNG
   // the same network as SCL:
   IF NOT #DONE AND (#UNICODE = WCHAR#'щ') THEN
       #ASCII_HEX := 16#F9;
       #DONE := TRUE;
   END_IF;
   IF NOT #DONE AND (#UNICODE = WCHAR#'ъ') THEN
       #ASCII_HEX := 16#FA;
       #DONE := TRUE;
   END_IF;
   IF NOT #DONE AND (#UNICODE = WCHAR#'ы') THEN
       #ASCII_HEX := 16#FB;
       #DONE := TRUE;
   END_IF;
   IF NOT #DONE AND (#UNICODE = WCHAR#'ь') THEN
       #ASCII_HEX := 16#FC;
       #DONE := TRUE;
   END_IF;
   IF NOT #DONE AND (#UNICODE = WCHAR#'э') THEN
       #ASCII_HEX := 16#FD;
       #DONE := TRUE;
   END_IF;
END_REGION

REGION Network 23: ю | я |
   RUNG wire#powerrail
      I_Contact( #DONE )
      { S7_Templates := "SrcType := WChar" } EQ_Contact(in1 := #UNICODE, in2 := WCHAR#'ю')
      Move(in := 16#FE, out1 => #ASCII_HEX)
      S_Coil( #DONE )
   END_RUNG
   RUNG wire#powerrail
      I_Contact( #DONE )
      { S7_Templates := "SrcType := WChar" } EQ_Contact(in1 := #UNICODE, in2 := WCHAR#'я')
      Move(in := 16#FF, out1 => #ASCII_HEX)
      S_Coil( #DONE )
   END_RUNG
   // the same network as SCL:
   IF NOT #DONE AND (#UNICODE = WCHAR#'ю') THEN
       #ASCII_HEX := 16#FE;
       #DONE := TRUE;
   END_IF;
   IF NOT #DONE AND (#UNICODE = WCHAR#'я') THEN
       #ASCII_HEX := 16#FF;
       #DONE := TRUE;
   END_IF;
END_REGION

REGION Network 24: A | B | C | D | E |
   RUNG wire#powerrail
      I_Contact( #DONE )
      { S7_Templates := "SrcType := WChar" } EQ_Contact(in1 := #UNICODE, in2 := WCHAR#'A')
      Move(in := 16#41, out1 => #ASCII_HEX)
      S_Coil( #DONE )
   END_RUNG
   RUNG wire#powerrail
      I_Contact( #DONE )
      { S7_Templates := "SrcType := WChar" } EQ_Contact(in1 := #UNICODE, in2 := WCHAR#'B')
      Move(in := 16#42, out1 => #ASCII_HEX)
      S_Coil( #DONE )
   END_RUNG
   RUNG wire#powerrail
      I_Contact( #DONE )
      { S7_Templates := "SrcType := WChar" } EQ_Contact(in1 := #UNICODE, in2 := WCHAR#'C')
      Move(in := 16#43, out1 => #ASCII_HEX)
      S_Coil( #DONE )
   END_RUNG
   RUNG wire#powerrail
      I_Contact( #DONE )
      { S7_Templates := "SrcType := WChar" } EQ_Contact(in1 := #UNICODE, in2 := WCHAR#'D')
      Move(in := 16#44, out1 => #ASCII_HEX)
      S_Coil( #DONE )
   END_RUNG
   RUNG wire#powerrail
      I_Contact( #DONE )
      { S7_Templates := "SrcType := WChar" } EQ_Contact(in1 := #UNICODE, in2 := WCHAR#'E')
      Move(in := 16#45, out1 => #ASCII_HEX)
      S_Coil( #DONE )
   END_RUNG
   // the same network as SCL:
   IF NOT #DONE AND (#UNICODE = WCHAR#'A') THEN
       #ASCII_HEX := 16#41;
       #DONE := TRUE;
   END_IF;
   IF NOT #DONE AND (#UNICODE = WCHAR#'B') THEN
       #ASCII_HEX := 16#42;
       #DONE := TRUE;
   END_IF;
   IF NOT #DONE AND (#UNICODE = WCHAR#'C') THEN
       #ASCII_HEX := 16#43;
       #DONE := TRUE;
   END_IF;
   IF NOT #DONE AND (#UNICODE = WCHAR#'D') THEN
       #ASCII_HEX := 16#44;
       #DONE := TRUE;
   END_IF;
   IF NOT #DONE AND (#UNICODE = WCHAR#'E') THEN
       #ASCII_HEX := 16#45;
       #DONE := TRUE;
   END_IF;
END_REGION

REGION Network 25: F | G | H | I | J |
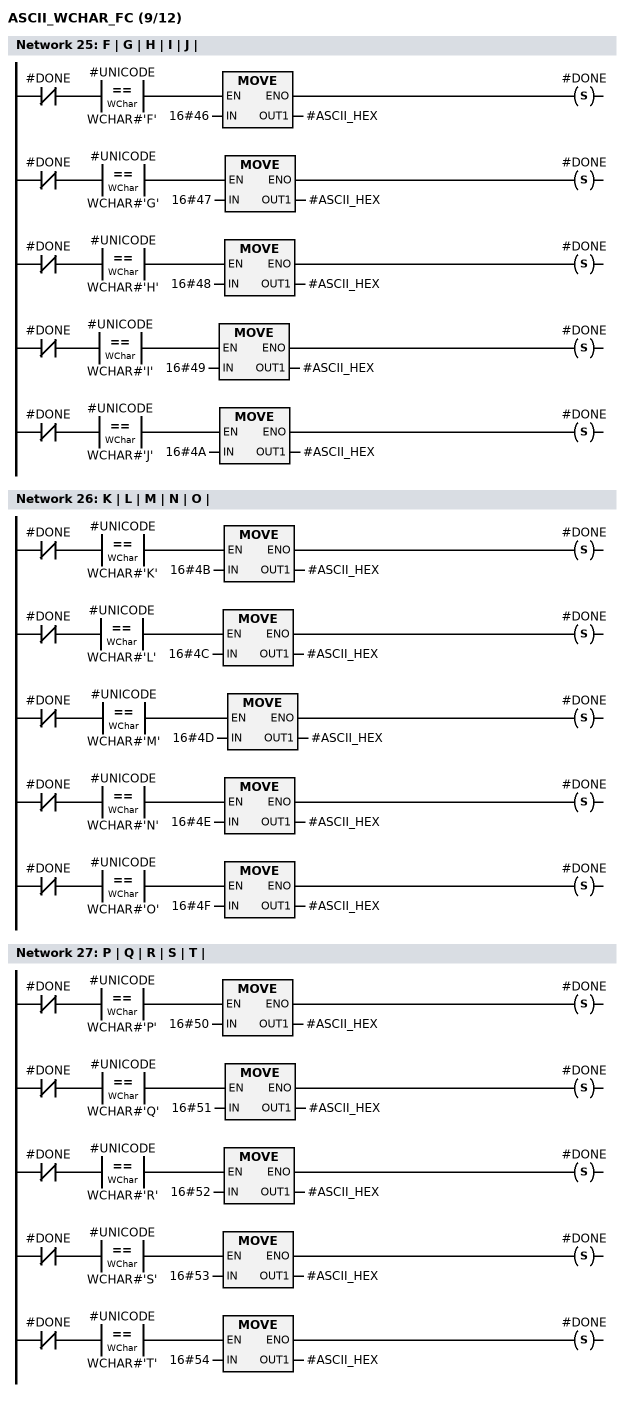
   RUNG wire#powerrail
      I_Contact( #DONE )
      { S7_Templates := "SrcType := WChar" } EQ_Contact(in1 := #UNICODE, in2 := WCHAR#'F')
      Move(in := 16#46, out1 => #ASCII_HEX)
      S_Coil( #DONE )
   END_RUNG
   RUNG wire#powerrail
      I_Contact( #DONE )
      { S7_Templates := "SrcType := WChar" } EQ_Contact(in1 := #UNICODE, in2 := WCHAR#'G')
      Move(in := 16#47, out1 => #ASCII_HEX)
      S_Coil( #DONE )
   END_RUNG
   RUNG wire#powerrail
      I_Contact( #DONE )
      { S7_Templates := "SrcType := WChar" } EQ_Contact(in1 := #UNICODE, in2 := WCHAR#'H')
      Move(in := 16#48, out1 => #ASCII_HEX)
      S_Coil( #DONE )
   END_RUNG
   RUNG wire#powerrail
      I_Contact( #DONE )
      { S7_Templates := "SrcType := WChar" } EQ_Contact(in1 := #UNICODE, in2 := WCHAR#'I')
      Move(in := 16#49, out1 => #ASCII_HEX)
      S_Coil( #DONE )
   END_RUNG
   RUNG wire#powerrail
      I_Contact( #DONE )
      { S7_Templates := "SrcType := WChar" } EQ_Contact(in1 := #UNICODE, in2 := WCHAR#'J')
      Move(in := 16#4A, out1 => #ASCII_HEX)
      S_Coil( #DONE )
   END_RUNG
   // the same network as SCL:
   IF NOT #DONE AND (#UNICODE = WCHAR#'F') THEN
       #ASCII_HEX := 16#46;
       #DONE := TRUE;
   END_IF;
   IF NOT #DONE AND (#UNICODE = WCHAR#'G') THEN
       #ASCII_HEX := 16#47;
       #DONE := TRUE;
   END_IF;
   IF NOT #DONE AND (#UNICODE = WCHAR#'H') THEN
       #ASCII_HEX := 16#48;
       #DONE := TRUE;
   END_IF;
   IF NOT #DONE AND (#UNICODE = WCHAR#'I') THEN
       #ASCII_HEX := 16#49;
       #DONE := TRUE;
   END_IF;
   IF NOT #DONE AND (#UNICODE = WCHAR#'J') THEN
       #ASCII_HEX := 16#4A;
       #DONE := TRUE;
   END_IF;
END_REGION

REGION Network 26: K | L | M | N | O |
   RUNG wire#powerrail
      I_Contact( #DONE )
      { S7_Templates := "SrcType := WChar" } EQ_Contact(in1 := #UNICODE, in2 := WCHAR#'K')
      Move(in := 16#4B, out1 => #ASCII_HEX)
      S_Coil( #DONE )
   END_RUNG
   RUNG wire#powerrail
      I_Contact( #DONE )
      { S7_Templates := "SrcType := WChar" } EQ_Contact(in1 := #UNICODE, in2 := WCHAR#'L')
      Move(in := 16#4C, out1 => #ASCII_HEX)
      S_Coil( #DONE )
   END_RUNG
   RUNG wire#powerrail
      I_Contact( #DONE )
      { S7_Templates := "SrcType := WChar" } EQ_Contact(in1 := #UNICODE, in2 := WCHAR#'M')
      Move(in := 16#4D, out1 => #ASCII_HEX)
      S_Coil( #DONE )
   END_RUNG
   RUNG wire#powerrail
      I_Contact( #DONE )
      { S7_Templates := "SrcType := WChar" } EQ_Contact(in1 := #UNICODE, in2 := WCHAR#'N')
      Move(in := 16#4E, out1 => #ASCII_HEX)
      S_Coil( #DONE )
   END_RUNG
   RUNG wire#powerrail
      I_Contact( #DONE )
      { S7_Templates := "SrcType := WChar" } EQ_Contact(in1 := #UNICODE, in2 := WCHAR#'O')
      Move(in := 16#4F, out1 => #ASCII_HEX)
      S_Coil( #DONE )
   END_RUNG
   // the same network as SCL:
   IF NOT #DONE AND (#UNICODE = WCHAR#'K') THEN
       #ASCII_HEX := 16#4B;
       #DONE := TRUE;
   END_IF;
   IF NOT #DONE AND (#UNICODE = WCHAR#'L') THEN
       #ASCII_HEX := 16#4C;
       #DONE := TRUE;
   END_IF;
   IF NOT #DONE AND (#UNICODE = WCHAR#'M') THEN
       #ASCII_HEX := 16#4D;
       #DONE := TRUE;
   END_IF;
   IF NOT #DONE AND (#UNICODE = WCHAR#'N') THEN
       #ASCII_HEX := 16#4E;
       #DONE := TRUE;
   END_IF;
   IF NOT #DONE AND (#UNICODE = WCHAR#'O') THEN
       #ASCII_HEX := 16#4F;
       #DONE := TRUE;
   END_IF;
END_REGION

REGION Network 27: P | Q | R | S | T |
   RUNG wire#powerrail
      I_Contact( #DONE )
      { S7_Templates := "SrcType := WChar" } EQ_Contact(in1 := #UNICODE, in2 := WCHAR#'P')
      Move(in := 16#50, out1 => #ASCII_HEX)
      S_Coil( #DONE )
   END_RUNG
   RUNG wire#powerrail
      I_Contact( #DONE )
      { S7_Templates := "SrcType := WChar" } EQ_Contact(in1 := #UNICODE, in2 := WCHAR#'Q')
      Move(in := 16#51, out1 => #ASCII_HEX)
      S_Coil( #DONE )
   END_RUNG
   RUNG wire#powerrail
      I_Contact( #DONE )
      { S7_Templates := "SrcType := WChar" } EQ_Contact(in1 := #UNICODE, in2 := WCHAR#'R')
      Move(in := 16#52, out1 => #ASCII_HEX)
      S_Coil( #DONE )
   END_RUNG
   RUNG wire#powerrail
      I_Contact( #DONE )
      { S7_Templates := "SrcType := WChar" } EQ_Contact(in1 := #UNICODE, in2 := WCHAR#'S')
      Move(in := 16#53, out1 => #ASCII_HEX)
      S_Coil( #DONE )
   END_RUNG
   RUNG wire#powerrail
      I_Contact( #DONE )
      { S7_Templates := "SrcType := WChar" } EQ_Contact(in1 := #UNICODE, in2 := WCHAR#'T')
      Move(in := 16#54, out1 => #ASCII_HEX)
      S_Coil( #DONE )
   END_RUNG
   // the same network as SCL:
   IF NOT #DONE AND (#UNICODE = WCHAR#'P') THEN
       #ASCII_HEX := 16#50;
       #DONE := TRUE;
   END_IF;
   IF NOT #DONE AND (#UNICODE = WCHAR#'Q') THEN
       #ASCII_HEX := 16#51;
       #DONE := TRUE;
   END_IF;
   IF NOT #DONE AND (#UNICODE = WCHAR#'R') THEN
       #ASCII_HEX := 16#52;
       #DONE := TRUE;
   END_IF;
   IF NOT #DONE AND (#UNICODE = WCHAR#'S') THEN
       #ASCII_HEX := 16#53;
       #DONE := TRUE;
   END_IF;
   IF NOT #DONE AND (#UNICODE = WCHAR#'T') THEN
       #ASCII_HEX := 16#54;
       #DONE := TRUE;
   END_IF;
END_REGION

REGION Network 28: U | V | W | X | Y | Z |
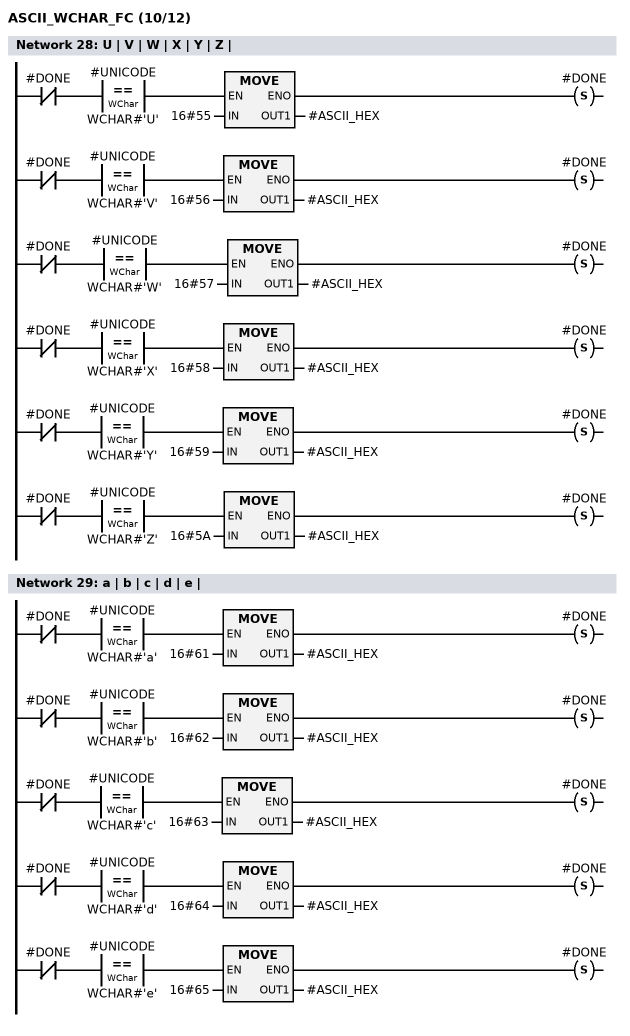
   RUNG wire#powerrail
      I_Contact( #DONE )
      { S7_Templates := "SrcType := WChar" } EQ_Contact(in1 := #UNICODE, in2 := WCHAR#'U')
      Move(in := 16#55, out1 => #ASCII_HEX)
      S_Coil( #DONE )
   END_RUNG
   RUNG wire#powerrail
      I_Contact( #DONE )
      { S7_Templates := "SrcType := WChar" } EQ_Contact(in1 := #UNICODE, in2 := WCHAR#'V')
      Move(in := 16#56, out1 => #ASCII_HEX)
      S_Coil( #DONE )
   END_RUNG
   RUNG wire#powerrail
      I_Contact( #DONE )
      { S7_Templates := "SrcType := WChar" } EQ_Contact(in1 := #UNICODE, in2 := WCHAR#'W')
      Move(in := 16#57, out1 => #ASCII_HEX)
      S_Coil( #DONE )
   END_RUNG
   RUNG wire#powerrail
      I_Contact( #DONE )
      { S7_Templates := "SrcType := WChar" } EQ_Contact(in1 := #UNICODE, in2 := WCHAR#'X')
      Move(in := 16#58, out1 => #ASCII_HEX)
      S_Coil( #DONE )
   END_RUNG
   RUNG wire#powerrail
      I_Contact( #DONE )
      { S7_Templates := "SrcType := WChar" } EQ_Contact(in1 := #UNICODE, in2 := WCHAR#'Y')
      Move(in := 16#59, out1 => #ASCII_HEX)
      S_Coil( #DONE )
   END_RUNG
   RUNG wire#powerrail
      I_Contact( #DONE )
      { S7_Templates := "SrcType := WChar" } EQ_Contact(in1 := #UNICODE, in2 := WCHAR#'Z')
      Move(in := 16#5A, out1 => #ASCII_HEX)
      S_Coil( #DONE )
   END_RUNG
   // the same network as SCL:
   IF NOT #DONE AND (#UNICODE = WCHAR#'U') THEN
       #ASCII_HEX := 16#55;
       #DONE := TRUE;
   END_IF;
   IF NOT #DONE AND (#UNICODE = WCHAR#'V') THEN
       #ASCII_HEX := 16#56;
       #DONE := TRUE;
   END_IF;
   IF NOT #DONE AND (#UNICODE = WCHAR#'W') THEN
       #ASCII_HEX := 16#57;
       #DONE := TRUE;
   END_IF;
   IF NOT #DONE AND (#UNICODE = WCHAR#'X') THEN
       #ASCII_HEX := 16#58;
       #DONE := TRUE;
   END_IF;
   IF NOT #DONE AND (#UNICODE = WCHAR#'Y') THEN
       #ASCII_HEX := 16#59;
       #DONE := TRUE;
   END_IF;
   IF NOT #DONE AND (#UNICODE = WCHAR#'Z') THEN
       #ASCII_HEX := 16#5A;
       #DONE := TRUE;
   END_IF;
END_REGION

REGION Network 29: a | b | c | d | e |
   RUNG wire#powerrail
      I_Contact( #DONE )
      { S7_Templates := "SrcType := WChar" } EQ_Contact(in1 := #UNICODE, in2 := WCHAR#'a')
      Move(in := 16#61, out1 => #ASCII_HEX)
      S_Coil( #DONE )
   END_RUNG
   RUNG wire#powerrail
      I_Contact( #DONE )
      { S7_Templates := "SrcType := WChar" } EQ_Contact(in1 := #UNICODE, in2 := WCHAR#'b')
      Move(in := 16#62, out1 => #ASCII_HEX)
      S_Coil( #DONE )
   END_RUNG
   RUNG wire#powerrail
      I_Contact( #DONE )
      { S7_Templates := "SrcType := WChar" } EQ_Contact(in1 := #UNICODE, in2 := WCHAR#'c')
      Move(in := 16#63, out1 => #ASCII_HEX)
      S_Coil( #DONE )
   END_RUNG
   RUNG wire#powerrail
      I_Contact( #DONE )
      { S7_Templates := "SrcType := WChar" } EQ_Contact(in1 := #UNICODE, in2 := WCHAR#'d')
      Move(in := 16#64, out1 => #ASCII_HEX)
      S_Coil( #DONE )
   END_RUNG
   RUNG wire#powerrail
      I_Contact( #DONE )
      { S7_Templates := "SrcType := WChar" } EQ_Contact(in1 := #UNICODE, in2 := WCHAR#'e')
      Move(in := 16#65, out1 => #ASCII_HEX)
      S_Coil( #DONE )
   END_RUNG
   // the same network as SCL:
   IF NOT #DONE AND (#UNICODE = WCHAR#'a') THEN
       #ASCII_HEX := 16#61;
       #DONE := TRUE;
   END_IF;
   IF NOT #DONE AND (#UNICODE = WCHAR#'b') THEN
       #ASCII_HEX := 16#62;
       #DONE := TRUE;
   END_IF;
   IF NOT #DONE AND (#UNICODE = WCHAR#'c') THEN
       #ASCII_HEX := 16#63;
       #DONE := TRUE;
   END_IF;
   IF NOT #DONE AND (#UNICODE = WCHAR#'d') THEN
       #ASCII_HEX := 16#64;
       #DONE := TRUE;
   END_IF;
   IF NOT #DONE AND (#UNICODE = WCHAR#'e') THEN
       #ASCII_HEX := 16#65;
       #DONE := TRUE;
   END_IF;
END_REGION

REGION Network 30: f | g | h | i | j |
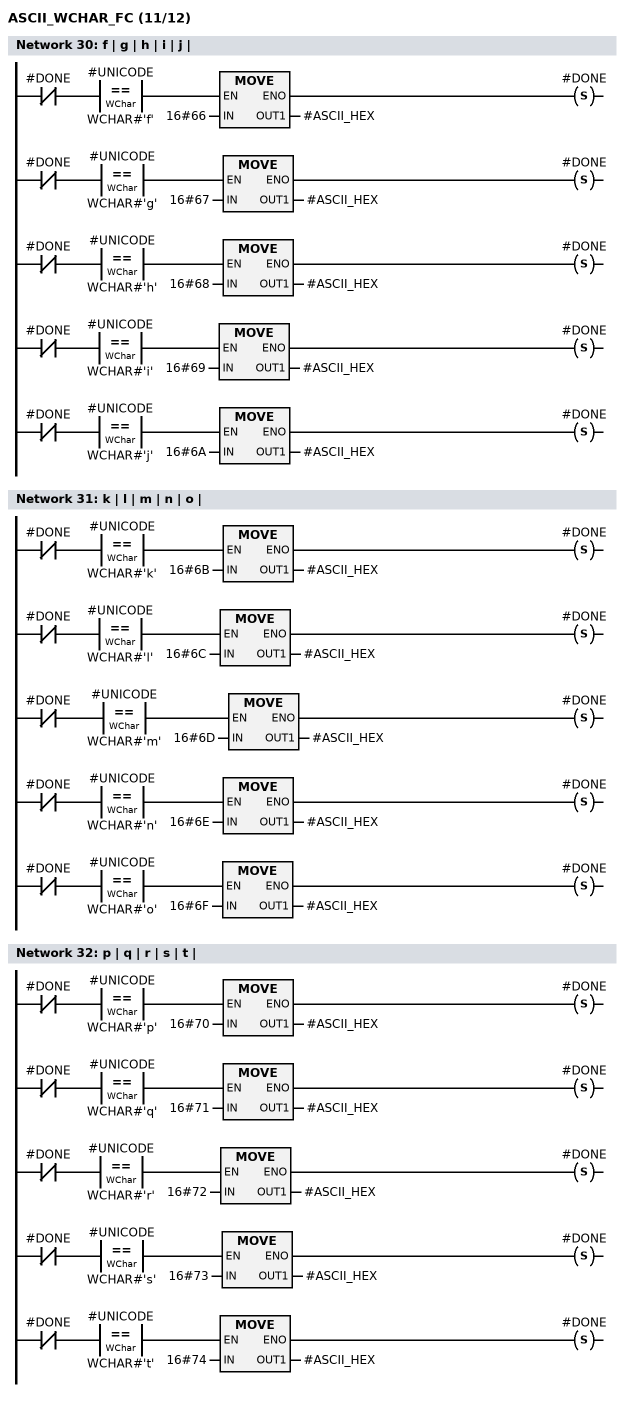
   RUNG wire#powerrail
      I_Contact( #DONE )
      { S7_Templates := "SrcType := WChar" } EQ_Contact(in1 := #UNICODE, in2 := WCHAR#'f')
      Move(in := 16#66, out1 => #ASCII_HEX)
      S_Coil( #DONE )
   END_RUNG
   RUNG wire#powerrail
      I_Contact( #DONE )
      { S7_Templates := "SrcType := WChar" } EQ_Contact(in1 := #UNICODE, in2 := WCHAR#'g')
      Move(in := 16#67, out1 => #ASCII_HEX)
      S_Coil( #DONE )
   END_RUNG
   RUNG wire#powerrail
      I_Contact( #DONE )
      { S7_Templates := "SrcType := WChar" } EQ_Contact(in1 := #UNICODE, in2 := WCHAR#'h')
      Move(in := 16#68, out1 => #ASCII_HEX)
      S_Coil( #DONE )
   END_RUNG
   RUNG wire#powerrail
      I_Contact( #DONE )
      { S7_Templates := "SrcType := WChar" } EQ_Contact(in1 := #UNICODE, in2 := WCHAR#'i')
      Move(in := 16#69, out1 => #ASCII_HEX)
      S_Coil( #DONE )
   END_RUNG
   RUNG wire#powerrail
      I_Contact( #DONE )
      { S7_Templates := "SrcType := WChar" } EQ_Contact(in1 := #UNICODE, in2 := WCHAR#'j')
      Move(in := 16#6A, out1 => #ASCII_HEX)
      S_Coil( #DONE )
   END_RUNG
   // the same network as SCL:
   IF NOT #DONE AND (#UNICODE = WCHAR#'f') THEN
       #ASCII_HEX := 16#66;
       #DONE := TRUE;
   END_IF;
   IF NOT #DONE AND (#UNICODE = WCHAR#'g') THEN
       #ASCII_HEX := 16#67;
       #DONE := TRUE;
   END_IF;
   IF NOT #DONE AND (#UNICODE = WCHAR#'h') THEN
       #ASCII_HEX := 16#68;
       #DONE := TRUE;
   END_IF;
   IF NOT #DONE AND (#UNICODE = WCHAR#'i') THEN
       #ASCII_HEX := 16#69;
       #DONE := TRUE;
   END_IF;
   IF NOT #DONE AND (#UNICODE = WCHAR#'j') THEN
       #ASCII_HEX := 16#6A;
       #DONE := TRUE;
   END_IF;
END_REGION

REGION Network 31: k | l | m | n | o |
   RUNG wire#powerrail
      I_Contact( #DONE )
      { S7_Templates := "SrcType := WChar" } EQ_Contact(in1 := #UNICODE, in2 := WCHAR#'k')
      Move(in := 16#6B, out1 => #ASCII_HEX)
      S_Coil( #DONE )
   END_RUNG
   RUNG wire#powerrail
      I_Contact( #DONE )
      { S7_Templates := "SrcType := WChar" } EQ_Contact(in1 := #UNICODE, in2 := WCHAR#'l')
      Move(in := 16#6C, out1 => #ASCII_HEX)
      S_Coil( #DONE )
   END_RUNG
   RUNG wire#powerrail
      I_Contact( #DONE )
      { S7_Templates := "SrcType := WChar" } EQ_Contact(in1 := #UNICODE, in2 := WCHAR#'m')
      Move(in := 16#6D, out1 => #ASCII_HEX)
      S_Coil( #DONE )
   END_RUNG
   RUNG wire#powerrail
      I_Contact( #DONE )
      { S7_Templates := "SrcType := WChar" } EQ_Contact(in1 := #UNICODE, in2 := WCHAR#'n')
      Move(in := 16#6E, out1 => #ASCII_HEX)
      S_Coil( #DONE )
   END_RUNG
   RUNG wire#powerrail
      I_Contact( #DONE )
      { S7_Templates := "SrcType := WChar" } EQ_Contact(in1 := #UNICODE, in2 := WCHAR#'o')
      Move(in := 16#6F, out1 => #ASCII_HEX)
      S_Coil( #DONE )
   END_RUNG
   // the same network as SCL:
   IF NOT #DONE AND (#UNICODE = WCHAR#'k') THEN
       #ASCII_HEX := 16#6B;
       #DONE := TRUE;
   END_IF;
   IF NOT #DONE AND (#UNICODE = WCHAR#'l') THEN
       #ASCII_HEX := 16#6C;
       #DONE := TRUE;
   END_IF;
   IF NOT #DONE AND (#UNICODE = WCHAR#'m') THEN
       #ASCII_HEX := 16#6D;
       #DONE := TRUE;
   END_IF;
   IF NOT #DONE AND (#UNICODE = WCHAR#'n') THEN
       #ASCII_HEX := 16#6E;
       #DONE := TRUE;
   END_IF;
   IF NOT #DONE AND (#UNICODE = WCHAR#'o') THEN
       #ASCII_HEX := 16#6F;
       #DONE := TRUE;
   END_IF;
END_REGION

REGION Network 32: p | q | r | s | t |
   RUNG wire#powerrail
      I_Contact( #DONE )
      { S7_Templates := "SrcType := WChar" } EQ_Contact(in1 := #UNICODE, in2 := WCHAR#'p')
      Move(in := 16#70, out1 => #ASCII_HEX)
      S_Coil( #DONE )
   END_RUNG
   RUNG wire#powerrail
      I_Contact( #DONE )
      { S7_Templates := "SrcType := WChar" } EQ_Contact(in1 := #UNICODE, in2 := WCHAR#'q')
      Move(in := 16#71, out1 => #ASCII_HEX)
      S_Coil( #DONE )
   END_RUNG
   RUNG wire#powerrail
      I_Contact( #DONE )
      { S7_Templates := "SrcType := WChar" } EQ_Contact(in1 := #UNICODE, in2 := WCHAR#'r')
      Move(in := 16#72, out1 => #ASCII_HEX)
      S_Coil( #DONE )
   END_RUNG
   RUNG wire#powerrail
      I_Contact( #DONE )
      { S7_Templates := "SrcType := WChar" } EQ_Contact(in1 := #UNICODE, in2 := WCHAR#'s')
      Move(in := 16#73, out1 => #ASCII_HEX)
      S_Coil( #DONE )
   END_RUNG
   RUNG wire#powerrail
      I_Contact( #DONE )
      { S7_Templates := "SrcType := WChar" } EQ_Contact(in1 := #UNICODE, in2 := WCHAR#'t')
      Move(in := 16#74, out1 => #ASCII_HEX)
      S_Coil( #DONE )
   END_RUNG
   // the same network as SCL:
   IF NOT #DONE AND (#UNICODE = WCHAR#'p') THEN
       #ASCII_HEX := 16#70;
       #DONE := TRUE;
   END_IF;
   IF NOT #DONE AND (#UNICODE = WCHAR#'q') THEN
       #ASCII_HEX := 16#71;
       #DONE := TRUE;
   END_IF;
   IF NOT #DONE AND (#UNICODE = WCHAR#'r') THEN
       #ASCII_HEX := 16#72;
       #DONE := TRUE;
   END_IF;
   IF NOT #DONE AND (#UNICODE = WCHAR#'s') THEN
       #ASCII_HEX := 16#73;
       #DONE := TRUE;
   END_IF;
   IF NOT #DONE AND (#UNICODE = WCHAR#'t') THEN
       #ASCII_HEX := 16#74;
       #DONE := TRUE;
   END_IF;
END_REGION

REGION Network 33: u | v | w | x | y | z |
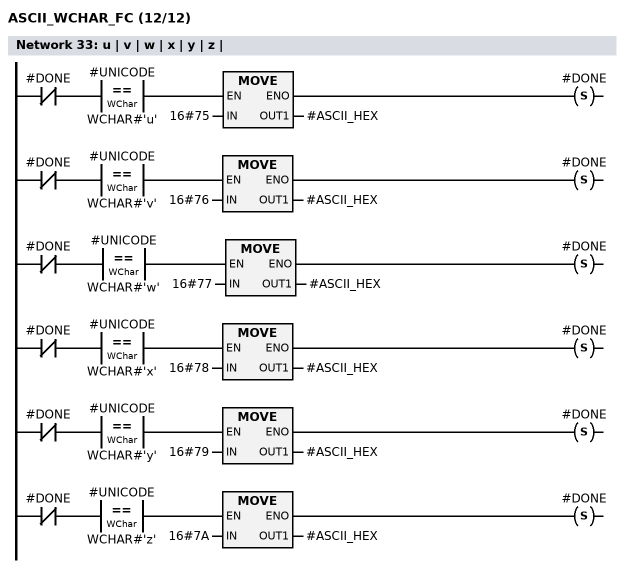
   RUNG wire#powerrail
      I_Contact( #DONE )
      { S7_Templates := "SrcType := WChar" } EQ_Contact(in1 := #UNICODE, in2 := WCHAR#'u')
      Move(in := 16#75, out1 => #ASCII_HEX)
      S_Coil( #DONE )
   END_RUNG
   RUNG wire#powerrail
      I_Contact( #DONE )
      { S7_Templates := "SrcType := WChar" } EQ_Contact(in1 := #UNICODE, in2 := WCHAR#'v')
      Move(in := 16#76, out1 => #ASCII_HEX)
      S_Coil( #DONE )
   END_RUNG
   RUNG wire#powerrail
      I_Contact( #DONE )
      { S7_Templates := "SrcType := WChar" } EQ_Contact(in1 := #UNICODE, in2 := WCHAR#'w')
      Move(in := 16#77, out1 => #ASCII_HEX)
      S_Coil( #DONE )
   END_RUNG
   RUNG wire#powerrail
      I_Contact( #DONE )
      { S7_Templates := "SrcType := WChar" } EQ_Contact(in1 := #UNICODE, in2 := WCHAR#'x')
      Move(in := 16#78, out1 => #ASCII_HEX)
      S_Coil( #DONE )
   END_RUNG
   RUNG wire#powerrail
      I_Contact( #DONE )
      { S7_Templates := "SrcType := WChar" } EQ_Contact(in1 := #UNICODE, in2 := WCHAR#'y')
      Move(in := 16#79, out1 => #ASCII_HEX)
      S_Coil( #DONE )
   END_RUNG
   RUNG wire#powerrail
      I_Contact( #DONE )
      { S7_Templates := "SrcType := WChar" } EQ_Contact(in1 := #UNICODE, in2 := WCHAR#'z')
      Move(in := 16#7A, out1 => #ASCII_HEX)
      S_Coil( #DONE )
   END_RUNG
   // the same network as SCL:
   IF NOT #DONE AND (#UNICODE = WCHAR#'u') THEN
       #ASCII_HEX := 16#75;
       #DONE := TRUE;
   END_IF;
   IF NOT #DONE AND (#UNICODE = WCHAR#'v') THEN
       #ASCII_HEX := 16#76;
       #DONE := TRUE;
   END_IF;
   IF NOT #DONE AND (#UNICODE = WCHAR#'w') THEN
       #ASCII_HEX := 16#77;
       #DONE := TRUE;
   END_IF;
   IF NOT #DONE AND (#UNICODE = WCHAR#'x') THEN
       #ASCII_HEX := 16#78;
       #DONE := TRUE;
   END_IF;
   IF NOT #DONE AND (#UNICODE = WCHAR#'y') THEN
       #ASCII_HEX := 16#79;
       #DONE := TRUE;
   END_IF;
   IF NOT #DONE AND (#UNICODE = WCHAR#'z') THEN
       #ASCII_HEX := 16#7A;
       #DONE := TRUE;
   END_IF;
END_REGION
END_FUNCTION
